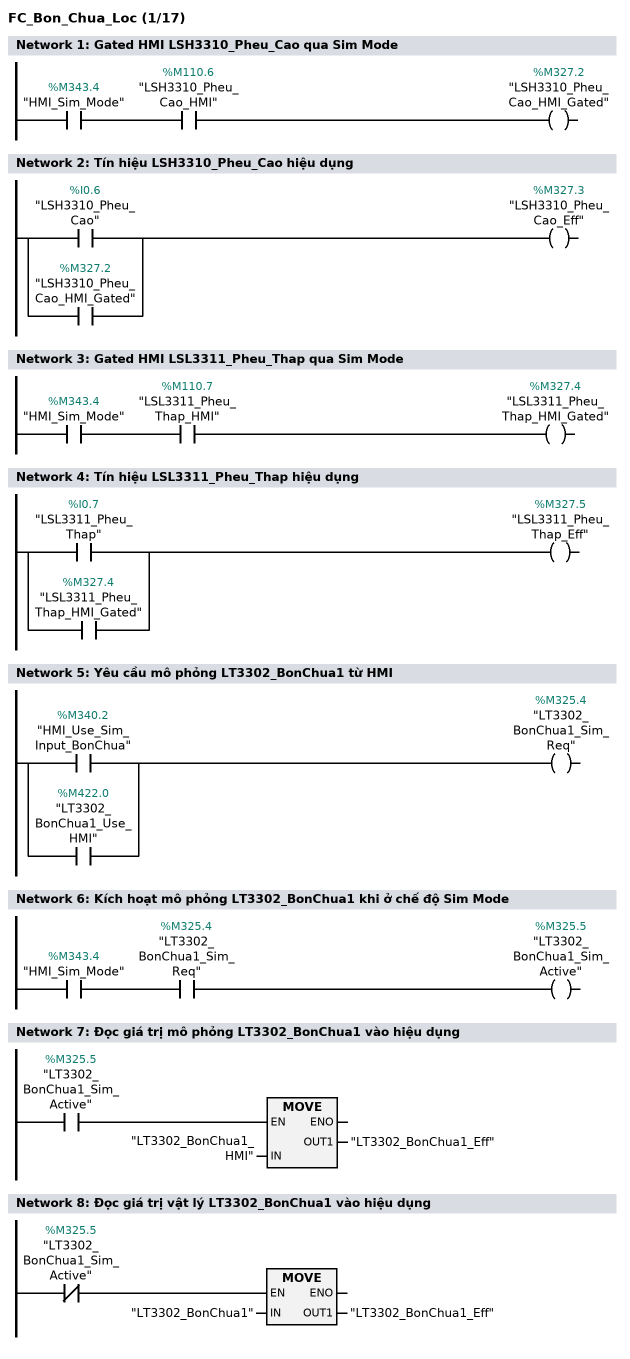
   RUNG wire#powerrail
      Contact( "HMI_Sim_Mode" )
      Contact( "LSH3310_Pheu_Cao_HMI" )
      Coil( "LSH3310_Pheu_Cao_HMI_Gated" )
   END_RUNG
   // the same network as SCL:
   "LSH3310_Pheu_Cao_HMI_Gated" := "HMI_Sim_Mode" AND "LSH3310_Pheu_Cao_HMI";
END_REGION

REGION Network 2: Tín hiệu LSH3310_Pheu_Cao hiệu dụng
   RUNG wire#powerrail
      Contact( "LSH3310_Pheu_Cao" )
      wire#w1
      Coil( "LSH3310_Pheu_Cao_Eff" )
   END_RUNG
   RUNG wire#powerrail
      Contact( "LSH3310_Pheu_Cao_HMI_Gated" )
   END_RUNG wire#w1
   // the same network as SCL:
   "LSH3310_Pheu_Cao_Eff" := "LSH3310_Pheu_Cao" OR "LSH3310_Pheu_Cao_HMI_Gated";
END_REGION

REGION Network 3: Gated HMI LSL3311_Pheu_Thap qua Sim Mode
   RUNG wire#powerrail
      Contact( "HMI_Sim_Mode" )
      Contact( "LSL3311_Pheu_Thap_HMI" )
      Coil( "LSL3311_Pheu_Thap_HMI_Gated" )
   END_RUNG
   // the same network as SCL:
   "LSL3311_Pheu_Thap_HMI_Gated" := "HMI_Sim_Mode" AND "LSL3311_Pheu_Thap_HMI";
END_REGION

REGION Network 4: Tín hiệu LSL3311_Pheu_Thap hiệu dụng
   RUNG wire#powerrail
      Contact( "LSL3311_Pheu_Thap" )
      wire#w1
      Coil( "LSL3311_Pheu_Thap_Eff" )
   END_RUNG
   RUNG wire#powerrail
      Contact( "LSL3311_Pheu_Thap_HMI_Gated" )
   END_RUNG wire#w1
   // the same network as SCL:
   "LSL3311_Pheu_Thap_Eff" := "LSL3311_Pheu_Thap" OR "LSL3311_Pheu_Thap_HMI_Gated";
END_REGION

REGION Network 5: Yêu cầu mô phỏng LT3302_BonChua1 từ HMI
   RUNG wire#powerrail
      Contact( "HMI_Use_Sim_Input_BonChua" )
      wire#w1
      Coil( "LT3302_BonChua1_Sim_Req" )
   END_RUNG
   RUNG wire#powerrail
      Contact( "LT3302_BonChua1_Use_HMI" )
   END_RUNG wire#w1
   // the same network as SCL:
   "LT3302_BonChua1_Sim_Req" := "HMI_Use_Sim_Input_BonChua" OR "LT3302_BonChua1_Use_HMI";
END_REGION

REGION Network 6: Kích hoạt mô phỏng LT3302_BonChua1 khi ở chế độ Sim Mode
   RUNG wire#powerrail
      Contact( "HMI_Sim_Mode" )
      Contact( "LT3302_BonChua1_Sim_Req" )
      Coil( "LT3302_BonChua1_Sim_Active" )
   END_RUNG
   // the same network as SCL:
   "LT3302_BonChua1_Sim_Active" := "HMI_Sim_Mode" AND "LT3302_BonChua1_Sim_Req";
END_REGION

REGION Network 7: Đọc giá trị mô phỏng LT3302_BonChua1 vào hiệu dụng
   RUNG wire#powerrail
      Contact( "LT3302_BonChua1_Sim_Active" )
      { S7_GenerateENO := "TRUE" } Move(in := "LT3302_BonChua1_HMI", out1 => "LT3302_BonChua1_Eff")
   END_RUNG
   // the same network as SCL:
   IF "LT3302_BonChua1_Sim_Active" THEN "LT3302_BonChua1_Eff" := "LT3302_BonChua1_HMI"; END_IF;
END_REGION

REGION Network 8: Đọc giá trị vật lý LT3302_BonChua1 vào hiệu dụng
   RUNG wire#powerrail
      I_Contact( "LT3302_BonChua1_Sim_Active" )
      { S7_GenerateENO := "TRUE" } Move(in := "LT3302_BonChua1", out1 => "LT3302_BonChua1_Eff")
   END_RUNG
   // the same network as SCL:
   IF NOT "LT3302_BonChua1_Sim_Active" THEN "LT3302_BonChua1_Eff" := "LT3302_BonChua1"; END_IF;
END_REGION

REGION Network 9: Yêu cầu mô phỏng TT3301_BonChua1 từ HMI
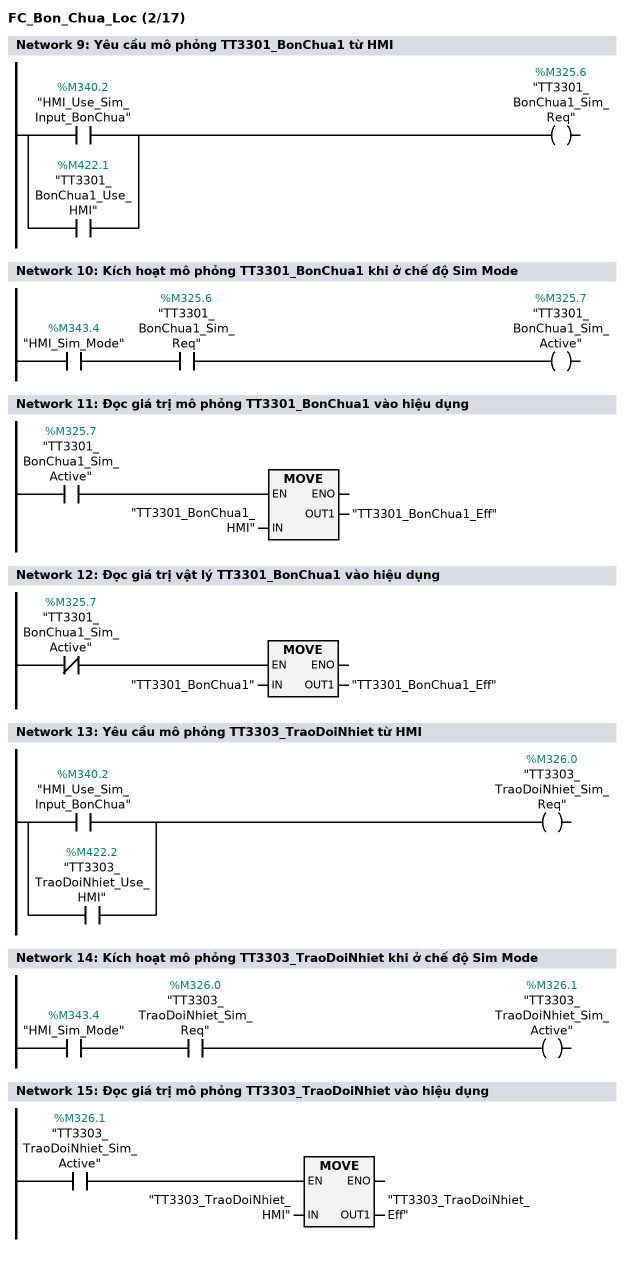
   RUNG wire#powerrail
      Contact( "HMI_Use_Sim_Input_BonChua" )
      wire#w1
      Coil( "TT3301_BonChua1_Sim_Req" )
   END_RUNG
   RUNG wire#powerrail
      Contact( "TT3301_BonChua1_Use_HMI" )
   END_RUNG wire#w1
   // the same network as SCL:
   "TT3301_BonChua1_Sim_Req" := "HMI_Use_Sim_Input_BonChua" OR "TT3301_BonChua1_Use_HMI";
END_REGION

REGION Network 10: Kích hoạt mô phỏng TT3301_BonChua1 khi ở chế độ Sim Mode
   RUNG wire#powerrail
      Contact( "HMI_Sim_Mode" )
      Contact( "TT3301_BonChua1_Sim_Req" )
      Coil( "TT3301_BonChua1_Sim_Active" )
   END_RUNG
   // the same network as SCL:
   "TT3301_BonChua1_Sim_Active" := "HMI_Sim_Mode" AND "TT3301_BonChua1_Sim_Req";
END_REGION

REGION Network 11: Đọc giá trị mô phỏng TT3301_BonChua1 vào hiệu dụng
   RUNG wire#powerrail
      Contact( "TT3301_BonChua1_Sim_Active" )
      { S7_GenerateENO := "TRUE" } Move(in := "TT3301_BonChua1_HMI", out1 => "TT3301_BonChua1_Eff")
   END_RUNG
   // the same network as SCL:
   IF "TT3301_BonChua1_Sim_Active" THEN "TT3301_BonChua1_Eff" := "TT3301_BonChua1_HMI"; END_IF;
END_REGION

REGION Network 12: Đọc giá trị vật lý TT3301_BonChua1 vào hiệu dụng
   RUNG wire#powerrail
      I_Contact( "TT3301_BonChua1_Sim_Active" )
      { S7_GenerateENO := "TRUE" } Move(in := "TT3301_BonChua1", out1 => "TT3301_BonChua1_Eff")
   END_RUNG
   // the same network as SCL:
   IF NOT "TT3301_BonChua1_Sim_Active" THEN "TT3301_BonChua1_Eff" := "TT3301_BonChua1"; END_IF;
END_REGION

REGION Network 13: Yêu cầu mô phỏng TT3303_TraoDoiNhiet từ HMI
   RUNG wire#powerrail
      Contact( "HMI_Use_Sim_Input_BonChua" )
      wire#w1
      Coil( "TT3303_TraoDoiNhiet_Sim_Req" )
   END_RUNG
   RUNG wire#powerrail
      Contact( "TT3303_TraoDoiNhiet_Use_HMI" )
   END_RUNG wire#w1
   // the same network as SCL:
   "TT3303_TraoDoiNhiet_Sim_Req" := "HMI_Use_Sim_Input_BonChua" OR "TT3303_TraoDoiNhiet_Use_HMI";
END_REGION

REGION Network 14: Kích hoạt mô phỏng TT3303_TraoDoiNhiet khi ở chế độ Sim Mode
   RUNG wire#powerrail
      Contact( "HMI_Sim_Mode" )
      Contact( "TT3303_TraoDoiNhiet_Sim_Req" )
      Coil( "TT3303_TraoDoiNhiet_Sim_Active" )
   END_RUNG
   // the same network as SCL:
   "TT3303_TraoDoiNhiet_Sim_Active" := "HMI_Sim_Mode" AND "TT3303_TraoDoiNhiet_Sim_Req";
END_REGION

REGION Network 15: Đọc giá trị mô phỏng TT3303_TraoDoiNhiet vào hiệu dụng
   RUNG wire#powerrail
      Contact( "TT3303_TraoDoiNhiet_Sim_Active" )
      { S7_GenerateENO := "TRUE" } Move(in := "TT3303_TraoDoiNhiet_HMI", out1 => "TT3303_TraoDoiNhiet_Eff")
   END_RUNG
   // the same network as SCL:
   IF "TT3303_TraoDoiNhiet_Sim_Active" THEN "TT3303_TraoDoiNhiet_Eff" := "TT3303_TraoDoiNhiet_HMI"; END_IF;
END_REGION

REGION Network 16: Đọc giá trị vật lý TT3303_TraoDoiNhiet vào hiệu dụng
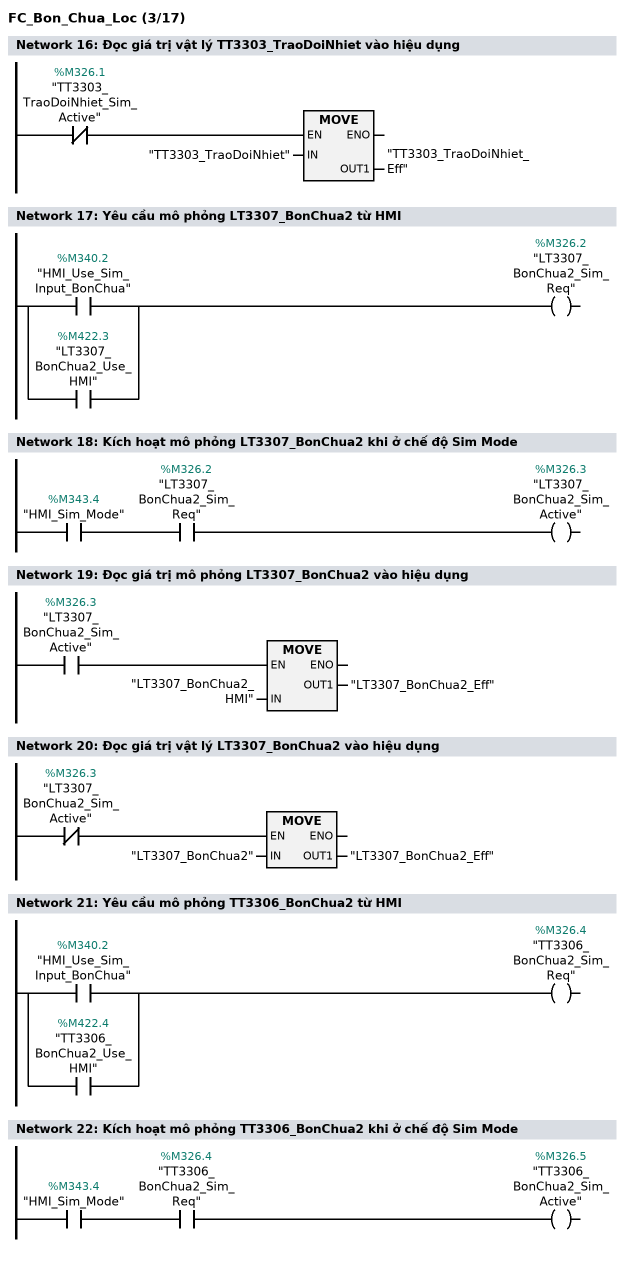
   RUNG wire#powerrail
      I_Contact( "TT3303_TraoDoiNhiet_Sim_Active" )
      { S7_GenerateENO := "TRUE" } Move(in := "TT3303_TraoDoiNhiet", out1 => "TT3303_TraoDoiNhiet_Eff")
   END_RUNG
   // the same network as SCL:
   IF NOT "TT3303_TraoDoiNhiet_Sim_Active" THEN "TT3303_TraoDoiNhiet_Eff" := "TT3303_TraoDoiNhiet"; END_IF;
END_REGION

REGION Network 17: Yêu cầu mô phỏng LT3307_BonChua2 từ HMI
   RUNG wire#powerrail
      Contact( "HMI_Use_Sim_Input_BonChua" )
      wire#w1
      Coil( "LT3307_BonChua2_Sim_Req" )
   END_RUNG
   RUNG wire#powerrail
      Contact( "LT3307_BonChua2_Use_HMI" )
   END_RUNG wire#w1
   // the same network as SCL:
   "LT3307_BonChua2_Sim_Req" := "HMI_Use_Sim_Input_BonChua" OR "LT3307_BonChua2_Use_HMI";
END_REGION

REGION Network 18: Kích hoạt mô phỏng LT3307_BonChua2 khi ở chế độ Sim Mode
   RUNG wire#powerrail
      Contact( "HMI_Sim_Mode" )
      Contact( "LT3307_BonChua2_Sim_Req" )
      Coil( "LT3307_BonChua2_Sim_Active" )
   END_RUNG
   // the same network as SCL:
   "LT3307_BonChua2_Sim_Active" := "HMI_Sim_Mode" AND "LT3307_BonChua2_Sim_Req";
END_REGION

REGION Network 19: Đọc giá trị mô phỏng LT3307_BonChua2 vào hiệu dụng
   RUNG wire#powerrail
      Contact( "LT3307_BonChua2_Sim_Active" )
      { S7_GenerateENO := "TRUE" } Move(in := "LT3307_BonChua2_HMI", out1 => "LT3307_BonChua2_Eff")
   END_RUNG
   // the same network as SCL:
   IF "LT3307_BonChua2_Sim_Active" THEN "LT3307_BonChua2_Eff" := "LT3307_BonChua2_HMI"; END_IF;
END_REGION

REGION Network 20: Đọc giá trị vật lý LT3307_BonChua2 vào hiệu dụng
   RUNG wire#powerrail
      I_Contact( "LT3307_BonChua2_Sim_Active" )
      { S7_GenerateENO := "TRUE" } Move(in := "LT3307_BonChua2", out1 => "LT3307_BonChua2_Eff")
   END_RUNG
   // the same network as SCL:
   IF NOT "LT3307_BonChua2_Sim_Active" THEN "LT3307_BonChua2_Eff" := "LT3307_BonChua2"; END_IF;
END_REGION

REGION Network 21: Yêu cầu mô phỏng TT3306_BonChua2 từ HMI
   RUNG wire#powerrail
      Contact( "HMI_Use_Sim_Input_BonChua" )
      wire#w1
      Coil( "TT3306_BonChua2_Sim_Req" )
   END_RUNG
   RUNG wire#powerrail
      Contact( "TT3306_BonChua2_Use_HMI" )
   END_RUNG wire#w1
   // the same network as SCL:
   "TT3306_BonChua2_Sim_Req" := "HMI_Use_Sim_Input_BonChua" OR "TT3306_BonChua2_Use_HMI";
END_REGION

REGION Network 22: Kích hoạt mô phỏng TT3306_BonChua2 khi ở chế độ Sim Mode
   RUNG wire#powerrail
      Contact( "HMI_Sim_Mode" )
      Contact( "TT3306_BonChua2_Sim_Req" )
      Coil( "TT3306_BonChua2_Sim_Active" )
   END_RUNG
   // the same network as SCL:
   "TT3306_BonChua2_Sim_Active" := "HMI_Sim_Mode" AND "TT3306_BonChua2_Sim_Req";
END_REGION

REGION Network 23: Đọc giá trị mô phỏng TT3306_BonChua2 vào hiệu dụng
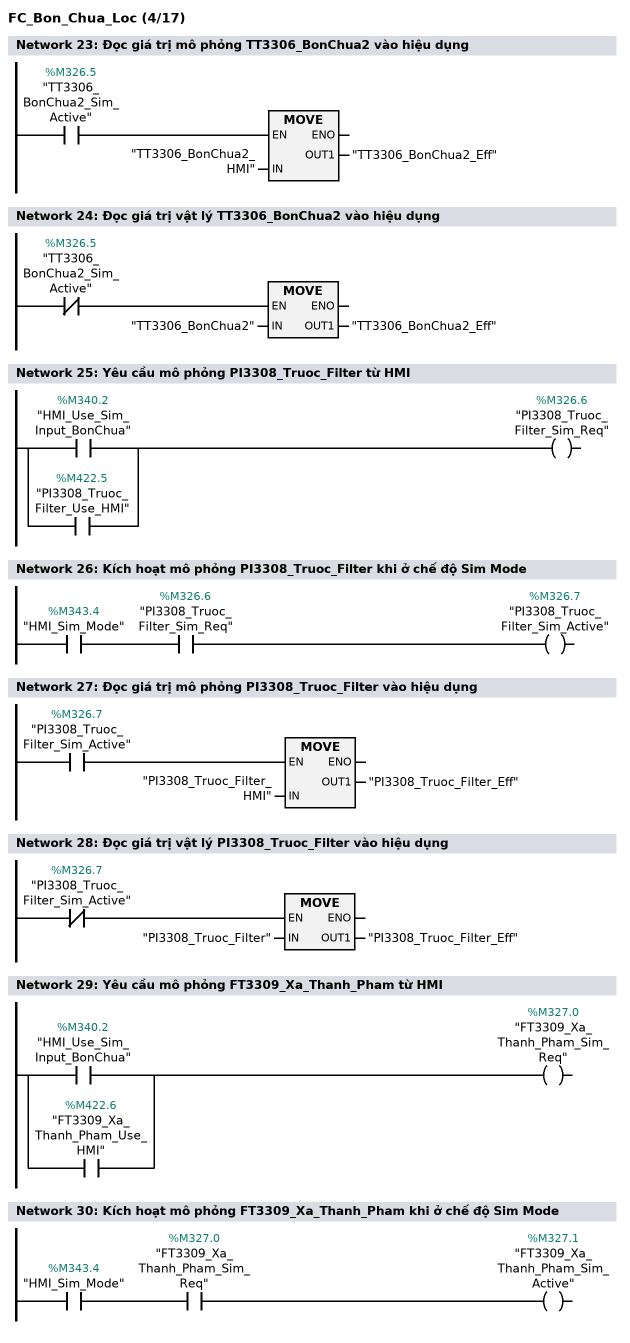
   RUNG wire#powerrail
      Contact( "TT3306_BonChua2_Sim_Active" )
      { S7_GenerateENO := "TRUE" } Move(in := "TT3306_BonChua2_HMI", out1 => "TT3306_BonChua2_Eff")
   END_RUNG
   // the same network as SCL:
   IF "TT3306_BonChua2_Sim_Active" THEN "TT3306_BonChua2_Eff" := "TT3306_BonChua2_HMI"; END_IF;
END_REGION

REGION Network 24: Đọc giá trị vật lý TT3306_BonChua2 vào hiệu dụng
   RUNG wire#powerrail
      I_Contact( "TT3306_BonChua2_Sim_Active" )
      { S7_GenerateENO := "TRUE" } Move(in := "TT3306_BonChua2", out1 => "TT3306_BonChua2_Eff")
   END_RUNG
   // the same network as SCL:
   IF NOT "TT3306_BonChua2_Sim_Active" THEN "TT3306_BonChua2_Eff" := "TT3306_BonChua2"; END_IF;
END_REGION

REGION Network 25: Yêu cầu mô phỏng PI3308_Truoc_Filter từ HMI
   RUNG wire#powerrail
      Contact( "HMI_Use_Sim_Input_BonChua" )
      wire#w1
      Coil( "PI3308_Truoc_Filter_Sim_Req" )
   END_RUNG
   RUNG wire#powerrail
      Contact( "PI3308_Truoc_Filter_Use_HMI" )
   END_RUNG wire#w1
   // the same network as SCL:
   "PI3308_Truoc_Filter_Sim_Req" := "HMI_Use_Sim_Input_BonChua" OR "PI3308_Truoc_Filter_Use_HMI";
END_REGION

REGION Network 26: Kích hoạt mô phỏng PI3308_Truoc_Filter khi ở chế độ Sim Mode
   RUNG wire#powerrail
      Contact( "HMI_Sim_Mode" )
      Contact( "PI3308_Truoc_Filter_Sim_Req" )
      Coil( "PI3308_Truoc_Filter_Sim_Active" )
   END_RUNG
   // the same network as SCL:
   "PI3308_Truoc_Filter_Sim_Active" := "HMI_Sim_Mode" AND "PI3308_Truoc_Filter_Sim_Req";
END_REGION

REGION Network 27: Đọc giá trị mô phỏng PI3308_Truoc_Filter vào hiệu dụng
   RUNG wire#powerrail
      Contact( "PI3308_Truoc_Filter_Sim_Active" )
      { S7_GenerateENO := "TRUE" } Move(in := "PI3308_Truoc_Filter_HMI", out1 => "PI3308_Truoc_Filter_Eff")
   END_RUNG
   // the same network as SCL:
   IF "PI3308_Truoc_Filter_Sim_Active" THEN "PI3308_Truoc_Filter_Eff" := "PI3308_Truoc_Filter_HMI"; END_IF;
END_REGION

REGION Network 28: Đọc giá trị vật lý PI3308_Truoc_Filter vào hiệu dụng
   RUNG wire#powerrail
      I_Contact( "PI3308_Truoc_Filter_Sim_Active" )
      { S7_GenerateENO := "TRUE" } Move(in := "PI3308_Truoc_Filter", out1 => "PI3308_Truoc_Filter_Eff")
   END_RUNG
   // the same network as SCL:
   IF NOT "PI3308_Truoc_Filter_Sim_Active" THEN "PI3308_Truoc_Filter_Eff" := "PI3308_Truoc_Filter"; END_IF;
END_REGION

REGION Network 29: Yêu cầu mô phỏng FT3309_Xa_Thanh_Pham từ HMI
   RUNG wire#powerrail
      Contact( "HMI_Use_Sim_Input_BonChua" )
      wire#w1
      Coil( "FT3309_Xa_Thanh_Pham_Sim_Req" )
   END_RUNG
   RUNG wire#powerrail
      Contact( "FT3309_Xa_Thanh_Pham_Use_HMI" )
   END_RUNG wire#w1
   // the same network as SCL:
   "FT3309_Xa_Thanh_Pham_Sim_Req" := "HMI_Use_Sim_Input_BonChua" OR "FT3309_Xa_Thanh_Pham_Use_HMI";
END_REGION

REGION Network 30: Kích hoạt mô phỏng FT3309_Xa_Thanh_Pham khi ở chế độ Sim Mode
   RUNG wire#powerrail
      Contact( "HMI_Sim_Mode" )
      Contact( "FT3309_Xa_Thanh_Pham_Sim_Req" )
      Coil( "FT3309_Xa_Thanh_Pham_Sim_Active" )
   END_RUNG
   // the same network as SCL:
   "FT3309_Xa_Thanh_Pham_Sim_Active" := "HMI_Sim_Mode" AND "FT3309_Xa_Thanh_Pham_Sim_Req";
END_REGION

REGION Network 31: Đọc giá trị mô phỏng FT3309_Xa_Thanh_Pham vào hiệu dụng
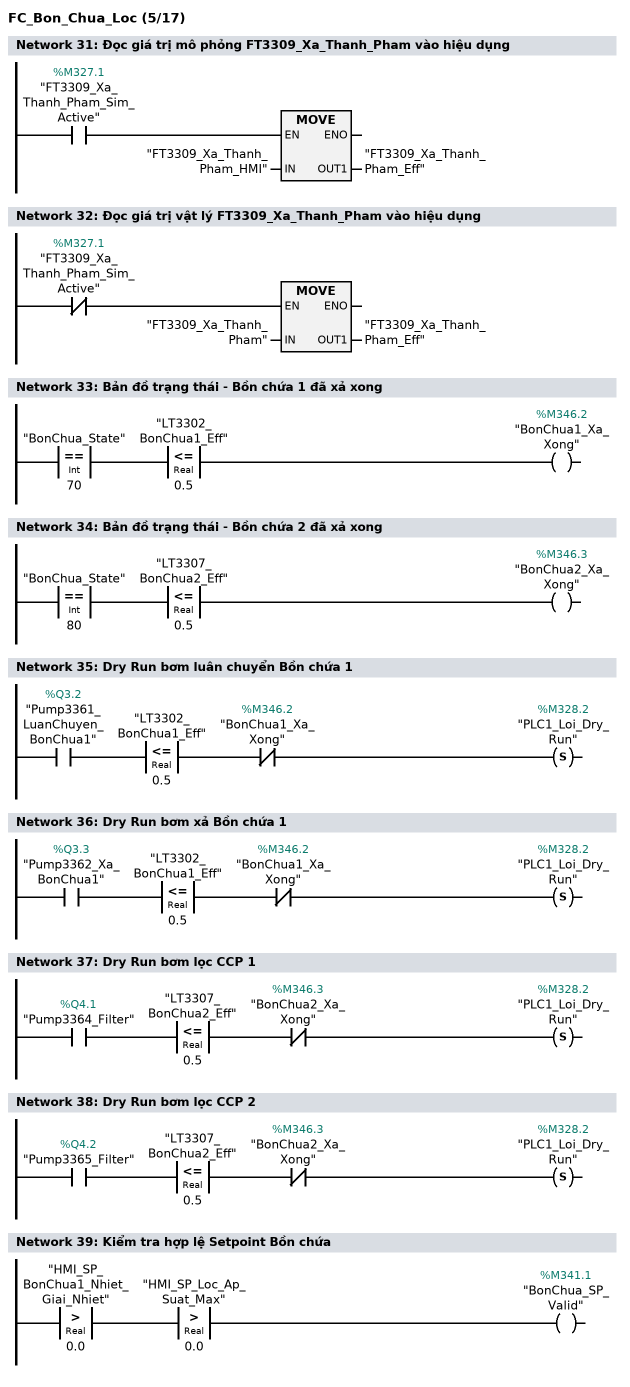
   RUNG wire#powerrail
      Contact( "FT3309_Xa_Thanh_Pham_Sim_Active" )
      { S7_GenerateENO := "TRUE" } Move(in := "FT3309_Xa_Thanh_Pham_HMI", out1 => "FT3309_Xa_Thanh_Pham_Eff")
   END_RUNG
   // the same network as SCL:
   IF "FT3309_Xa_Thanh_Pham_Sim_Active" THEN
       "FT3309_Xa_Thanh_Pham_Eff" := "FT3309_Xa_Thanh_Pham_HMI";
   END_IF;
END_REGION

REGION Network 32: Đọc giá trị vật lý FT3309_Xa_Thanh_Pham vào hiệu dụng
   RUNG wire#powerrail
      I_Contact( "FT3309_Xa_Thanh_Pham_Sim_Active" )
      { S7_GenerateENO := "TRUE" } Move(in := "FT3309_Xa_Thanh_Pham", out1 => "FT3309_Xa_Thanh_Pham_Eff")
   END_RUNG
   // the same network as SCL:
   IF NOT "FT3309_Xa_Thanh_Pham_Sim_Active" THEN
       "FT3309_Xa_Thanh_Pham_Eff" := "FT3309_Xa_Thanh_Pham";
   END_IF;
END_REGION

REGION Network 33: Bản đồ trạng thái - Bồn chứa 1 đã xả xong
   RUNG wire#powerrail
      { S7_Templates := "SrcType := Int" } EQ_Contact(in1 := "BonChua_State", in2 := 70)
      { S7_Templates := "SrcType := Real" } LE_Contact(in1 := "LT3302_BonChua1_Eff", in2 := 0.5)
      Coil( "BonChua1_Xa_Xong" )
   END_RUNG
   // the same network as SCL:
   "BonChua1_Xa_Xong" := ("BonChua_State" = 70) AND ("LT3302_BonChua1_Eff" <= 0.5);
END_REGION

REGION Network 34: Bản đồ trạng thái - Bồn chứa 2 đã xả xong
   RUNG wire#powerrail
      { S7_Templates := "SrcType := Int" } EQ_Contact(in1 := "BonChua_State", in2 := 80)
      { S7_Templates := "SrcType := Real" } LE_Contact(in1 := "LT3307_BonChua2_Eff", in2 := 0.5)
      Coil( "BonChua2_Xa_Xong" )
   END_RUNG
   // the same network as SCL:
   "BonChua2_Xa_Xong" := ("BonChua_State" = 80) AND ("LT3307_BonChua2_Eff" <= 0.5);
END_REGION

REGION Network 35: Dry Run bơm luân chuyển Bồn chứa 1
   RUNG wire#powerrail
      Contact( "Pump3361_LuanChuyen_BonChua1" )
      { S7_Templates := "SrcType := Real" } LE_Contact(in1 := "LT3302_BonChua1_Eff", in2 := 0.5)
      I_Contact( "BonChua1_Xa_Xong" )
      S_Coil( "PLC1_Loi_Dry_Run" )
   END_RUNG
   // the same network as SCL:
   IF "Pump3361_LuanChuyen_BonChua1" AND ("LT3302_BonChua1_Eff" <= 0.5) AND NOT "BonChua1_Xa_Xong" THEN
       "PLC1_Loi_Dry_Run" := TRUE;
   END_IF;
END_REGION

REGION Network 36: Dry Run bơm xả Bồn chứa 1
   RUNG wire#powerrail
      Contact( "Pump3362_Xa_BonChua1" )
      { S7_Templates := "SrcType := Real" } LE_Contact(in1 := "LT3302_BonChua1_Eff", in2 := 0.5)
      I_Contact( "BonChua1_Xa_Xong" )
      S_Coil( "PLC1_Loi_Dry_Run" )
   END_RUNG
   // the same network as SCL:
   IF "Pump3362_Xa_BonChua1" AND ("LT3302_BonChua1_Eff" <= 0.5) AND NOT "BonChua1_Xa_Xong" THEN
       "PLC1_Loi_Dry_Run" := TRUE;
   END_IF;
END_REGION

REGION Network 37: Dry Run bơm lọc CCP 1
   RUNG wire#powerrail
      Contact( "Pump3364_Filter" )
      { S7_Templates := "SrcType := Real" } LE_Contact(in1 := "LT3307_BonChua2_Eff", in2 := 0.5)
      I_Contact( "BonChua2_Xa_Xong" )
      S_Coil( "PLC1_Loi_Dry_Run" )
   END_RUNG
   // the same network as SCL:
   IF "Pump3364_Filter" AND ("LT3307_BonChua2_Eff" <= 0.5) AND NOT "BonChua2_Xa_Xong" THEN
       "PLC1_Loi_Dry_Run" := TRUE;
   END_IF;
END_REGION

REGION Network 38: Dry Run bơm lọc CCP 2
   RUNG wire#powerrail
      Contact( "Pump3365_Filter" )
      { S7_Templates := "SrcType := Real" } LE_Contact(in1 := "LT3307_BonChua2_Eff", in2 := 0.5)
      I_Contact( "BonChua2_Xa_Xong" )
      S_Coil( "PLC1_Loi_Dry_Run" )
   END_RUNG
   // the same network as SCL:
   IF "Pump3365_Filter" AND ("LT3307_BonChua2_Eff" <= 0.5) AND NOT "BonChua2_Xa_Xong" THEN
       "PLC1_Loi_Dry_Run" := TRUE;
   END_IF;
END_REGION

REGION Network 39: Kiểm tra hợp lệ Setpoint Bồn chứa
   RUNG wire#powerrail
      { S7_Templates := "SrcType := Real" } GT_Contact(in1 := "HMI_SP_BonChua1_Nhiet_Giai_Nhiet", in2 := 0.0)
      { S7_Templates := "SrcType := Real" } GT_Contact(in1 := "HMI_SP_Loc_Ap_Suat_Max", in2 := 0.0)
      Coil( "BonChua_SP_Valid" )
   END_RUNG
   // the same network as SCL:
   "BonChua_SP_Valid" := ("HMI_SP_BonChua1_Nhiet_Giai_Nhiet" > 0.0) AND ("HMI_SP_Loc_Ap_Suat_Max" > 0.0);
END_REGION

REGION Network 40: Stop hoặc Lỗi tổng - reset BonChua_Step_Nhan_Dich
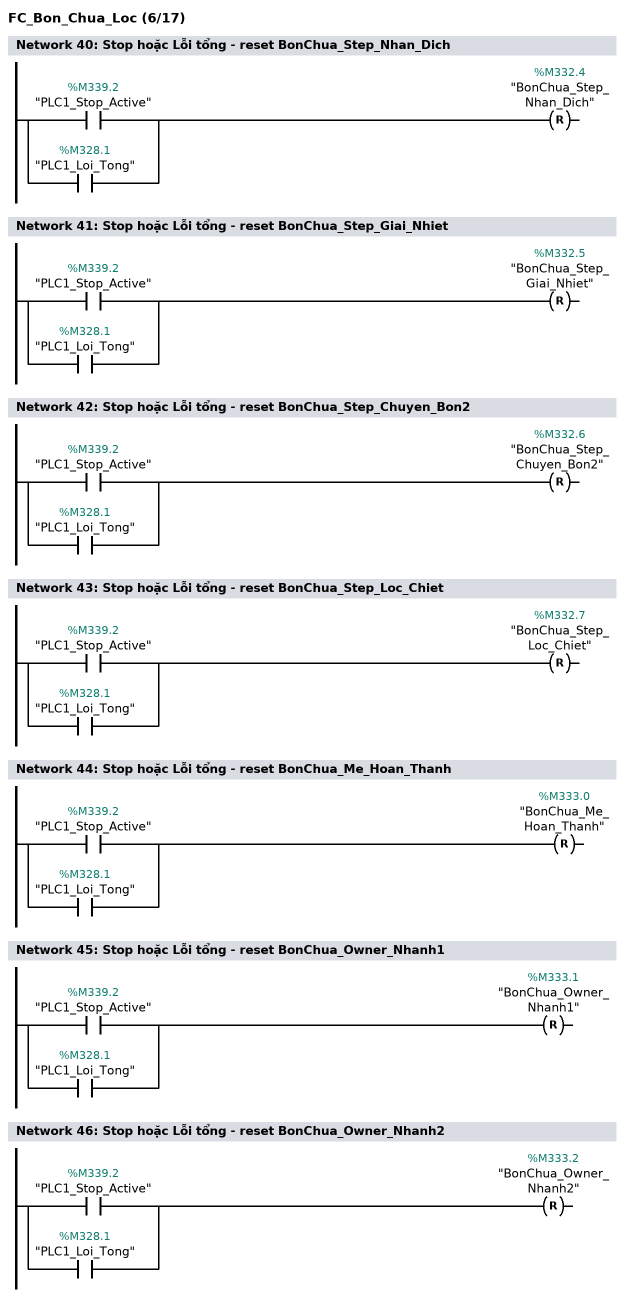
   RUNG wire#powerrail
      Contact( "PLC1_Stop_Active" )
      wire#w1
      R_Coil( "BonChua_Step_Nhan_Dich" )
   END_RUNG
   RUNG wire#powerrail
      Contact( "PLC1_Loi_Tong" )
   END_RUNG wire#w1
   // the same network as SCL:
   IF "PLC1_Stop_Active" OR "PLC1_Loi_Tong" THEN "BonChua_Step_Nhan_Dich" := FALSE; END_IF;
END_REGION

REGION Network 41: Stop hoặc Lỗi tổng - reset BonChua_Step_Giai_Nhiet
   RUNG wire#powerrail
      Contact( "PLC1_Stop_Active" )
      wire#w1
      R_Coil( "BonChua_Step_Giai_Nhiet" )
   END_RUNG
   RUNG wire#powerrail
      Contact( "PLC1_Loi_Tong" )
   END_RUNG wire#w1
   // the same network as SCL:
   IF "PLC1_Stop_Active" OR "PLC1_Loi_Tong" THEN "BonChua_Step_Giai_Nhiet" := FALSE; END_IF;
END_REGION

REGION Network 42: Stop hoặc Lỗi tổng - reset BonChua_Step_Chuyen_Bon2
   RUNG wire#powerrail
      Contact( "PLC1_Stop_Active" )
      wire#w1
      R_Coil( "BonChua_Step_Chuyen_Bon2" )
   END_RUNG
   RUNG wire#powerrail
      Contact( "PLC1_Loi_Tong" )
   END_RUNG wire#w1
   // the same network as SCL:
   IF "PLC1_Stop_Active" OR "PLC1_Loi_Tong" THEN "BonChua_Step_Chuyen_Bon2" := FALSE; END_IF;
END_REGION

REGION Network 43: Stop hoặc Lỗi tổng - reset BonChua_Step_Loc_Chiet
   RUNG wire#powerrail
      Contact( "PLC1_Stop_Active" )
      wire#w1
      R_Coil( "BonChua_Step_Loc_Chiet" )
   END_RUNG
   RUNG wire#powerrail
      Contact( "PLC1_Loi_Tong" )
   END_RUNG wire#w1
   // the same network as SCL:
   IF "PLC1_Stop_Active" OR "PLC1_Loi_Tong" THEN "BonChua_Step_Loc_Chiet" := FALSE; END_IF;
END_REGION

REGION Network 44: Stop hoặc Lỗi tổng - reset BonChua_Me_Hoan_Thanh
   RUNG wire#powerrail
      Contact( "PLC1_Stop_Active" )
      wire#w1
      R_Coil( "BonChua_Me_Hoan_Thanh" )
   END_RUNG
   RUNG wire#powerrail
      Contact( "PLC1_Loi_Tong" )
   END_RUNG wire#w1
   // the same network as SCL:
   IF "PLC1_Stop_Active" OR "PLC1_Loi_Tong" THEN "BonChua_Me_Hoan_Thanh" := FALSE; END_IF;
END_REGION

REGION Network 45: Stop hoặc Lỗi tổng - reset BonChua_Owner_Nhanh1
   RUNG wire#powerrail
      Contact( "PLC1_Stop_Active" )
      wire#w1
      R_Coil( "BonChua_Owner_Nhanh1" )
   END_RUNG
   RUNG wire#powerrail
      Contact( "PLC1_Loi_Tong" )
   END_RUNG wire#w1
   // the same network as SCL:
   IF "PLC1_Stop_Active" OR "PLC1_Loi_Tong" THEN "BonChua_Owner_Nhanh1" := FALSE; END_IF;
END_REGION

REGION Network 46: Stop hoặc Lỗi tổng - reset BonChua_Owner_Nhanh2
   RUNG wire#powerrail
      Contact( "PLC1_Stop_Active" )
      wire#w1
      R_Coil( "BonChua_Owner_Nhanh2" )
   END_RUNG
   RUNG wire#powerrail
      Contact( "PLC1_Loi_Tong" )
   END_RUNG wire#w1
   // the same network as SCL:
   IF "PLC1_Stop_Active" OR "PLC1_Loi_Tong" THEN "BonChua_Owner_Nhanh2" := FALSE; END_IF;
END_REGION

REGION Network 47: Stop hoặc Lỗi tổng - reset V3331_Xa_BonChua1
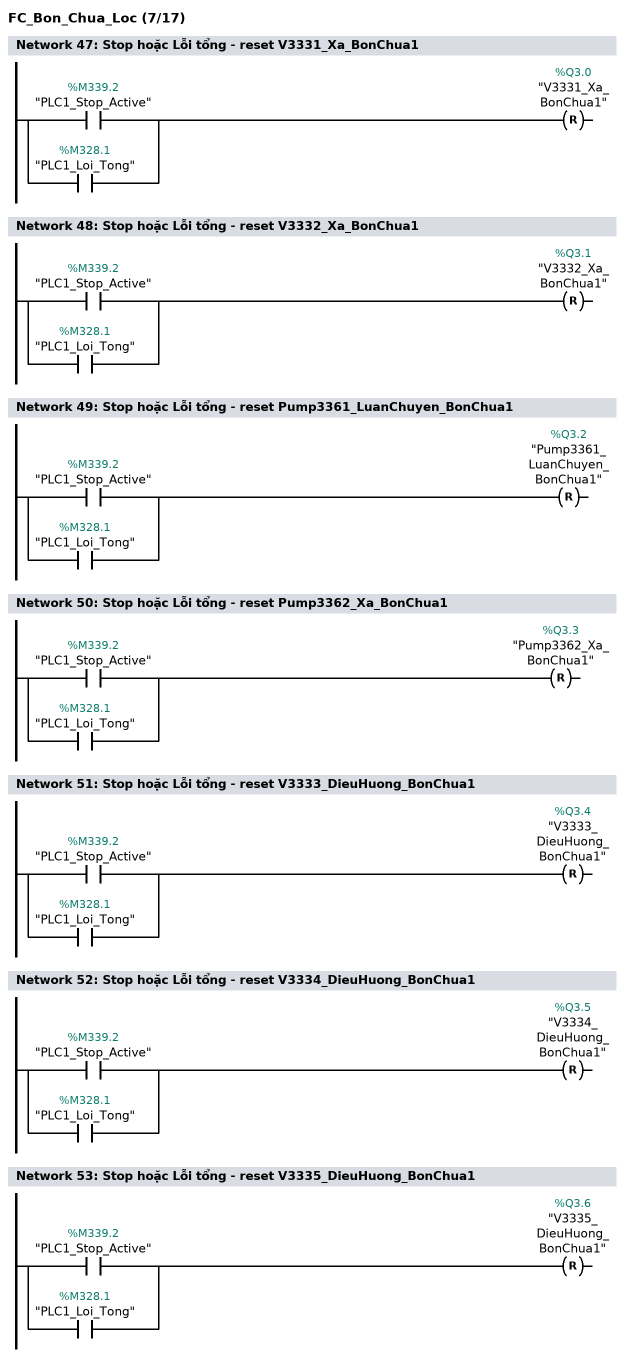
   RUNG wire#powerrail
      Contact( "PLC1_Stop_Active" )
      wire#w1
      R_Coil( "V3331_Xa_BonChua1" )
   END_RUNG
   RUNG wire#powerrail
      Contact( "PLC1_Loi_Tong" )
   END_RUNG wire#w1
   // the same network as SCL:
   IF "PLC1_Stop_Active" OR "PLC1_Loi_Tong" THEN "V3331_Xa_BonChua1" := FALSE; END_IF;
END_REGION

REGION Network 48: Stop hoặc Lỗi tổng - reset V3332_Xa_BonChua1
   RUNG wire#powerrail
      Contact( "PLC1_Stop_Active" )
      wire#w1
      R_Coil( "V3332_Xa_BonChua1" )
   END_RUNG
   RUNG wire#powerrail
      Contact( "PLC1_Loi_Tong" )
   END_RUNG wire#w1
   // the same network as SCL:
   IF "PLC1_Stop_Active" OR "PLC1_Loi_Tong" THEN "V3332_Xa_BonChua1" := FALSE; END_IF;
END_REGION

REGION Network 49: Stop hoặc Lỗi tổng - reset Pump3361_LuanChuyen_BonChua1
   RUNG wire#powerrail
      Contact( "PLC1_Stop_Active" )
      wire#w1
      R_Coil( "Pump3361_LuanChuyen_BonChua1" )
   END_RUNG
   RUNG wire#powerrail
      Contact( "PLC1_Loi_Tong" )
   END_RUNG wire#w1
   // the same network as SCL:
   IF "PLC1_Stop_Active" OR "PLC1_Loi_Tong" THEN "Pump3361_LuanChuyen_BonChua1" := FALSE; END_IF;
END_REGION

REGION Network 50: Stop hoặc Lỗi tổng - reset Pump3362_Xa_BonChua1
   RUNG wire#powerrail
      Contact( "PLC1_Stop_Active" )
      wire#w1
      R_Coil( "Pump3362_Xa_BonChua1" )
   END_RUNG
   RUNG wire#powerrail
      Contact( "PLC1_Loi_Tong" )
   END_RUNG wire#w1
   // the same network as SCL:
   IF "PLC1_Stop_Active" OR "PLC1_Loi_Tong" THEN "Pump3362_Xa_BonChua1" := FALSE; END_IF;
END_REGION

REGION Network 51: Stop hoặc Lỗi tổng - reset V3333_DieuHuong_BonChua1
   RUNG wire#powerrail
      Contact( "PLC1_Stop_Active" )
      wire#w1
      R_Coil( "V3333_DieuHuong_BonChua1" )
   END_RUNG
   RUNG wire#powerrail
      Contact( "PLC1_Loi_Tong" )
   END_RUNG wire#w1
   // the same network as SCL:
   IF "PLC1_Stop_Active" OR "PLC1_Loi_Tong" THEN "V3333_DieuHuong_BonChua1" := FALSE; END_IF;
END_REGION

REGION Network 52: Stop hoặc Lỗi tổng - reset V3334_DieuHuong_BonChua1
   RUNG wire#powerrail
      Contact( "PLC1_Stop_Active" )
      wire#w1
      R_Coil( "V3334_DieuHuong_BonChua1" )
   END_RUNG
   RUNG wire#powerrail
      Contact( "PLC1_Loi_Tong" )
   END_RUNG wire#w1
   // the same network as SCL:
   IF "PLC1_Stop_Active" OR "PLC1_Loi_Tong" THEN "V3334_DieuHuong_BonChua1" := FALSE; END_IF;
END_REGION

REGION Network 53: Stop hoặc Lỗi tổng - reset V3335_DieuHuong_BonChua1
   RUNG wire#powerrail
      Contact( "PLC1_Stop_Active" )
      wire#w1
      R_Coil( "V3335_DieuHuong_BonChua1" )
   END_RUNG
   RUNG wire#powerrail
      Contact( "PLC1_Loi_Tong" )
   END_RUNG wire#w1
   // the same network as SCL:
   IF "PLC1_Stop_Active" OR "PLC1_Loi_Tong" THEN "V3335_DieuHuong_BonChua1" := FALSE; END_IF;
END_REGION

REGION Network 54: Stop hoặc Lỗi tổng - reset V3338_Xa_BonChua2
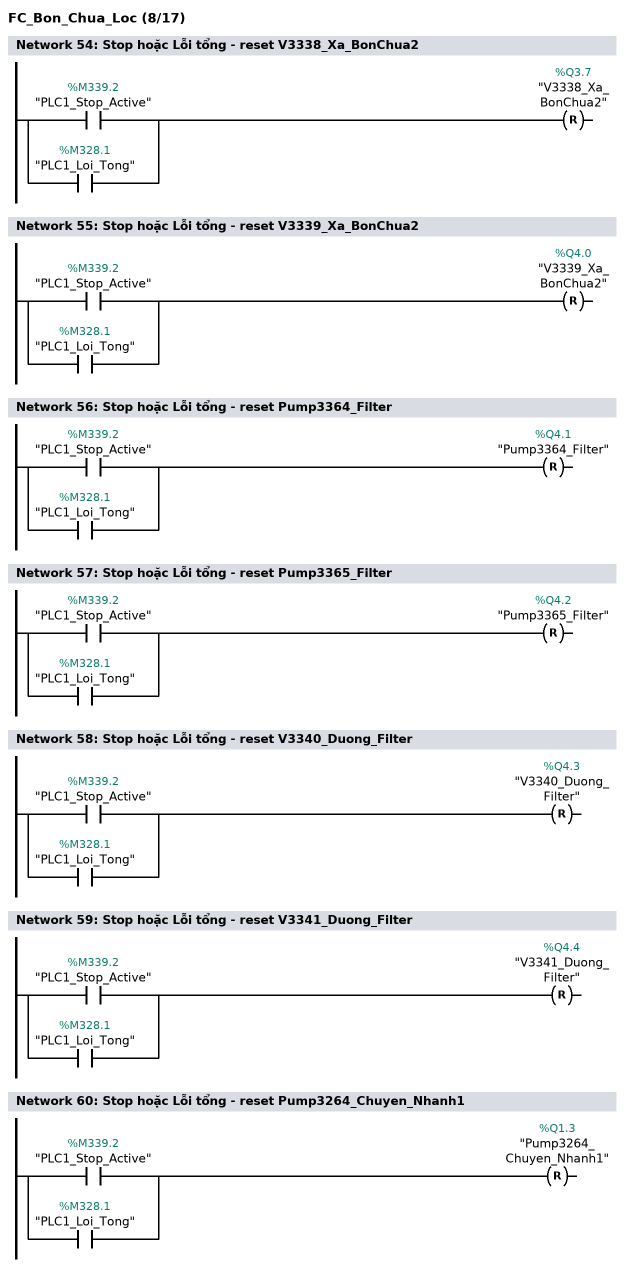
   RUNG wire#powerrail
      Contact( "PLC1_Stop_Active" )
      wire#w1
      R_Coil( "V3338_Xa_BonChua2" )
   END_RUNG
   RUNG wire#powerrail
      Contact( "PLC1_Loi_Tong" )
   END_RUNG wire#w1
   // the same network as SCL:
   IF "PLC1_Stop_Active" OR "PLC1_Loi_Tong" THEN "V3338_Xa_BonChua2" := FALSE; END_IF;
END_REGION

REGION Network 55: Stop hoặc Lỗi tổng - reset V3339_Xa_BonChua2
   RUNG wire#powerrail
      Contact( "PLC1_Stop_Active" )
      wire#w1
      R_Coil( "V3339_Xa_BonChua2" )
   END_RUNG
   RUNG wire#powerrail
      Contact( "PLC1_Loi_Tong" )
   END_RUNG wire#w1
   // the same network as SCL:
   IF "PLC1_Stop_Active" OR "PLC1_Loi_Tong" THEN "V3339_Xa_BonChua2" := FALSE; END_IF;
END_REGION

REGION Network 56: Stop hoặc Lỗi tổng - reset Pump3364_Filter
   RUNG wire#powerrail
      Contact( "PLC1_Stop_Active" )
      wire#w1
      R_Coil( "Pump3364_Filter" )
   END_RUNG
   RUNG wire#powerrail
      Contact( "PLC1_Loi_Tong" )
   END_RUNG wire#w1
   // the same network as SCL:
   IF "PLC1_Stop_Active" OR "PLC1_Loi_Tong" THEN "Pump3364_Filter" := FALSE; END_IF;
END_REGION

REGION Network 57: Stop hoặc Lỗi tổng - reset Pump3365_Filter
   RUNG wire#powerrail
      Contact( "PLC1_Stop_Active" )
      wire#w1
      R_Coil( "Pump3365_Filter" )
   END_RUNG
   RUNG wire#powerrail
      Contact( "PLC1_Loi_Tong" )
   END_RUNG wire#w1
   // the same network as SCL:
   IF "PLC1_Stop_Active" OR "PLC1_Loi_Tong" THEN "Pump3365_Filter" := FALSE; END_IF;
END_REGION

REGION Network 58: Stop hoặc Lỗi tổng - reset V3340_Duong_Filter
   RUNG wire#powerrail
      Contact( "PLC1_Stop_Active" )
      wire#w1
      R_Coil( "V3340_Duong_Filter" )
   END_RUNG
   RUNG wire#powerrail
      Contact( "PLC1_Loi_Tong" )
   END_RUNG wire#w1
   // the same network as SCL:
   IF "PLC1_Stop_Active" OR "PLC1_Loi_Tong" THEN "V3340_Duong_Filter" := FALSE; END_IF;
END_REGION

REGION Network 59: Stop hoặc Lỗi tổng - reset V3341_Duong_Filter
   RUNG wire#powerrail
      Contact( "PLC1_Stop_Active" )
      wire#w1
      R_Coil( "V3341_Duong_Filter" )
   END_RUNG
   RUNG wire#powerrail
      Contact( "PLC1_Loi_Tong" )
   END_RUNG wire#w1
   // the same network as SCL:
   IF "PLC1_Stop_Active" OR "PLC1_Loi_Tong" THEN "V3341_Duong_Filter" := FALSE; END_IF;
END_REGION

REGION Network 60: Stop hoặc Lỗi tổng - reset Pump3264_Chuyen_Nhanh1
   RUNG wire#powerrail
      Contact( "PLC1_Stop_Active" )
      wire#w1
      R_Coil( "Pump3264_Chuyen_Nhanh1" )
   END_RUNG
   RUNG wire#powerrail
      Contact( "PLC1_Loi_Tong" )
   END_RUNG wire#w1
   // the same network as SCL:
   IF "PLC1_Stop_Active" OR "PLC1_Loi_Tong" THEN "Pump3264_Chuyen_Nhanh1" := FALSE; END_IF;
END_REGION

REGION Network 61: Stop hoặc Lỗi tổng - reset Pump3265_Chuyen_Nhanh2_Cmd
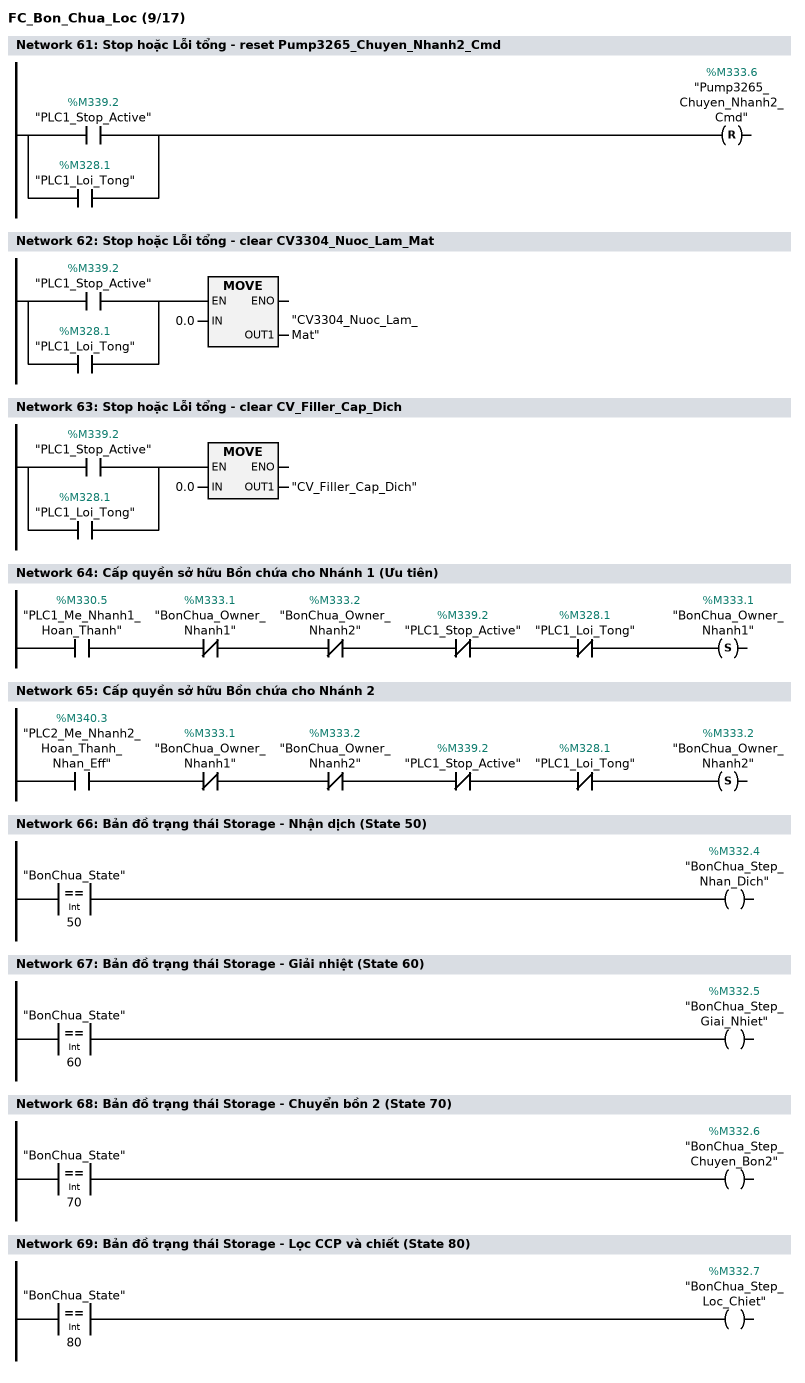
   RUNG wire#powerrail
      Contact( "PLC1_Stop_Active" )
      wire#w1
      R_Coil( "Pump3265_Chuyen_Nhanh2_Cmd" )
   END_RUNG
   RUNG wire#powerrail
      Contact( "PLC1_Loi_Tong" )
   END_RUNG wire#w1
   // the same network as SCL:
   IF "PLC1_Stop_Active" OR "PLC1_Loi_Tong" THEN "Pump3265_Chuyen_Nhanh2_Cmd" := FALSE; END_IF;
END_REGION

REGION Network 62: Stop hoặc Lỗi tổng - clear CV3304_Nuoc_Lam_Mat
   RUNG wire#powerrail
      Contact( "PLC1_Stop_Active" )
      wire#w1
      { S7_GenerateENO := "TRUE" } Move(in := 0.0, out1 => "CV3304_Nuoc_Lam_Mat")
   END_RUNG
   RUNG wire#powerrail
      Contact( "PLC1_Loi_Tong" )
   END_RUNG wire#w1
   // the same network as SCL:
   IF "PLC1_Stop_Active" OR "PLC1_Loi_Tong" THEN "CV3304_Nuoc_Lam_Mat" := 0.0; END_IF;
END_REGION

REGION Network 63: Stop hoặc Lỗi tổng - clear CV_Filler_Cap_Dich
   RUNG wire#powerrail
      Contact( "PLC1_Stop_Active" )
      wire#w1
      { S7_GenerateENO := "TRUE" } Move(in := 0.0, out1 => "CV_Filler_Cap_Dich")
   END_RUNG
   RUNG wire#powerrail
      Contact( "PLC1_Loi_Tong" )
   END_RUNG wire#w1
   // the same network as SCL:
   IF "PLC1_Stop_Active" OR "PLC1_Loi_Tong" THEN "CV_Filler_Cap_Dich" := 0.0; END_IF;
END_REGION

REGION Network 64: Cấp quyền sở hữu Bồn chứa cho Nhánh 1 (Ưu tiên)
   RUNG wire#powerrail
      Contact( "PLC1_Me_Nhanh1_Hoan_Thanh" )
      I_Contact( "BonChua_Owner_Nhanh1" )
      I_Contact( "BonChua_Owner_Nhanh2" )
      I_Contact( "PLC1_Stop_Active" )
      I_Contact( "PLC1_Loi_Tong" )
      S_Coil( "BonChua_Owner_Nhanh1" )
   END_RUNG
   // the same network as SCL:
   IF "PLC1_Me_Nhanh1_Hoan_Thanh" AND NOT "BonChua_Owner_Nhanh1" AND NOT "BonChua_Owner_Nhanh2" AND NOT "PLC1_Stop_Active" AND NOT "PLC1_Loi_Tong" THEN
       "BonChua_Owner_Nhanh1" := TRUE;
   END_IF;
END_REGION

REGION Network 65: Cấp quyền sở hữu Bồn chứa cho Nhánh 2
   RUNG wire#powerrail
      Contact( "PLC2_Me_Nhanh2_Hoan_Thanh_Nhan_Eff" )
      I_Contact( "BonChua_Owner_Nhanh1" )
      I_Contact( "BonChua_Owner_Nhanh2" )
      I_Contact( "PLC1_Stop_Active" )
      I_Contact( "PLC1_Loi_Tong" )
      S_Coil( "BonChua_Owner_Nhanh2" )
   END_RUNG
   // the same network as SCL:
   IF "PLC2_Me_Nhanh2_Hoan_Thanh_Nhan_Eff" AND NOT "BonChua_Owner_Nhanh1" AND NOT "BonChua_Owner_Nhanh2" AND NOT "PLC1_Stop_Active" AND NOT "PLC1_Loi_Tong" THEN
       "BonChua_Owner_Nhanh2" := TRUE;
   END_IF;
END_REGION

REGION Network 66: Bản đồ trạng thái Storage - Nhận dịch (State 50)
   RUNG wire#powerrail
      { S7_Templates := "SrcType := Int" } EQ_Contact(in1 := "BonChua_State", in2 := 50)
      Coil( "BonChua_Step_Nhan_Dich" )
   END_RUNG
   // the same network as SCL:
   "BonChua_Step_Nhan_Dich" := "BonChua_State" = 50;
END_REGION

REGION Network 67: Bản đồ trạng thái Storage - Giải nhiệt (State 60)
   RUNG wire#powerrail
      { S7_Templates := "SrcType := Int" } EQ_Contact(in1 := "BonChua_State", in2 := 60)
      Coil( "BonChua_Step_Giai_Nhiet" )
   END_RUNG
   // the same network as SCL:
   "BonChua_Step_Giai_Nhiet" := "BonChua_State" = 60;
END_REGION

REGION Network 68: Bản đồ trạng thái Storage - Chuyển bồn 2 (State 70)
   RUNG wire#powerrail
      { S7_Templates := "SrcType := Int" } EQ_Contact(in1 := "BonChua_State", in2 := 70)
      Coil( "BonChua_Step_Chuyen_Bon2" )
   END_RUNG
   // the same network as SCL:
   "BonChua_Step_Chuyen_Bon2" := "BonChua_State" = 70;
END_REGION

REGION Network 69: Bản đồ trạng thái Storage - Lọc CCP và chiết (State 80)
   RUNG wire#powerrail
      { S7_Templates := "SrcType := Int" } EQ_Contact(in1 := "BonChua_State", in2 := 80)
      Coil( "BonChua_Step_Loc_Chiet" )
   END_RUNG
   // the same network as SCL:
   "BonChua_Step_Loc_Chiet" := "BonChua_State" = 80;
END_REGION

REGION Network 70: Nhận mẻ từ Nhánh 1 hoặc Nhánh 2 thành công - Chuyển sang State 50
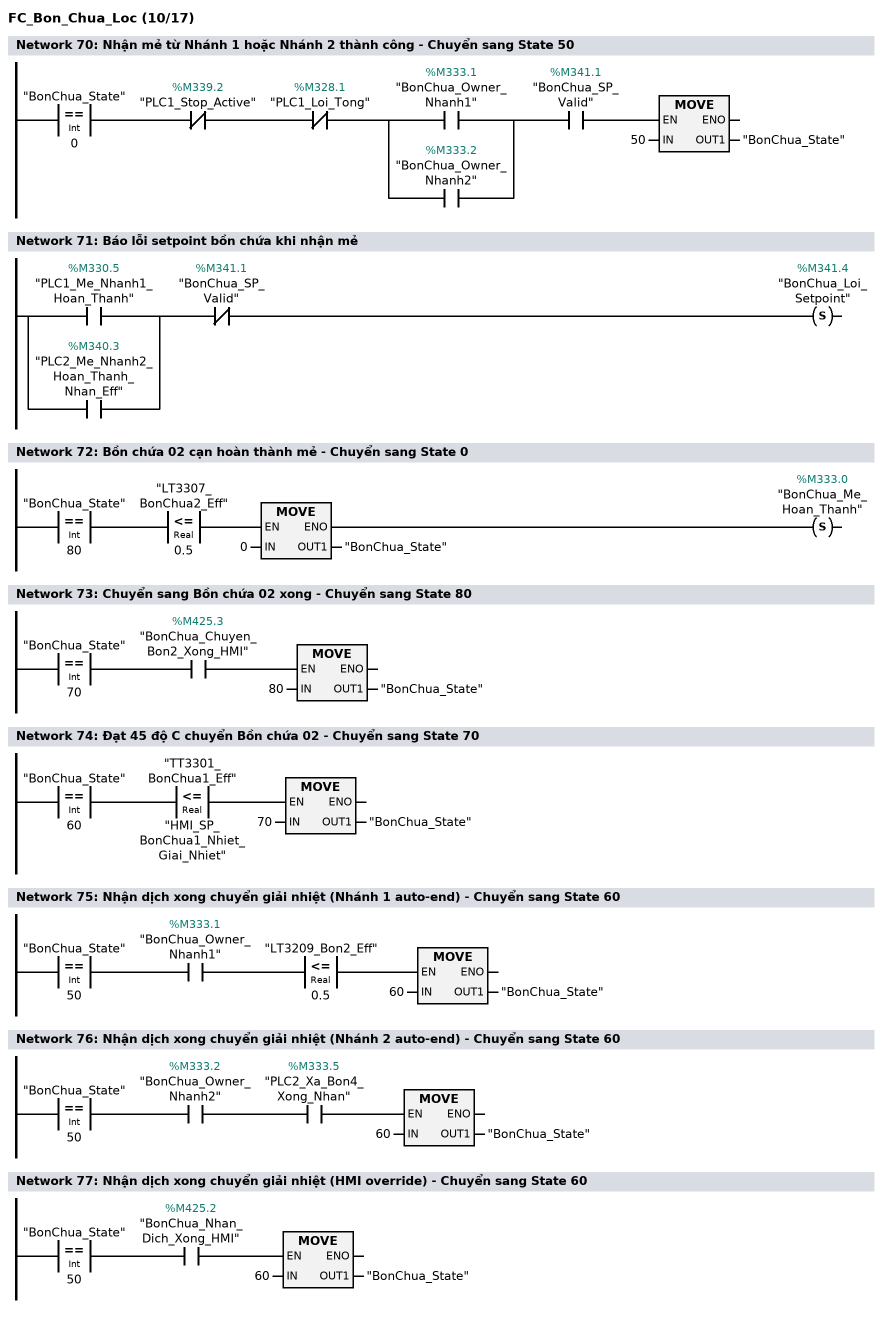
   RUNG wire#powerrail
      { S7_Templates := "SrcType := Int" } EQ_Contact(in1 := "BonChua_State", in2 := 0)
      I_Contact( "PLC1_Stop_Active" )
      I_Contact( "PLC1_Loi_Tong" )
      wire#w1
      Contact( "BonChua_Owner_Nhanh1" )
      wire#w2
      Contact( "BonChua_SP_Valid" )
      { S7_GenerateENO := "TRUE" } Move(in := 50, out1 => "BonChua_State")
   END_RUNG
   RUNG wire#w1
      Contact( "BonChua_Owner_Nhanh2" )
   END_RUNG wire#w2
   // the same network as SCL:
   IF ("BonChua_State" = 0) AND NOT "PLC1_Stop_Active" AND NOT "PLC1_Loi_Tong" AND ("BonChua_Owner_Nhanh1" OR "BonChua_Owner_Nhanh2") AND "BonChua_SP_Valid" THEN
       "BonChua_State" := 50;
   END_IF;
END_REGION

REGION Network 71: Báo lỗi setpoint bồn chứa khi nhận mẻ
   RUNG wire#powerrail
      Contact( "PLC1_Me_Nhanh1_Hoan_Thanh" )
      wire#w1
      I_Contact( "BonChua_SP_Valid" )
      S_Coil( "BonChua_Loi_Setpoint" )
   END_RUNG
   RUNG wire#powerrail
      Contact( "PLC2_Me_Nhanh2_Hoan_Thanh_Nhan_Eff" )
   END_RUNG wire#w1
   // the same network as SCL:
   IF ("PLC1_Me_Nhanh1_Hoan_Thanh" OR "PLC2_Me_Nhanh2_Hoan_Thanh_Nhan_Eff") AND NOT "BonChua_SP_Valid" THEN
       "BonChua_Loi_Setpoint" := TRUE;
   END_IF;
END_REGION

REGION Network 72: Bồn chứa 02 cạn hoàn thành mẻ - Chuyển sang State 0
   RUNG wire#powerrail
      { S7_Templates := "SrcType := Int" } EQ_Contact(in1 := "BonChua_State", in2 := 80)
      { S7_Templates := "SrcType := Real" } LE_Contact(in1 := "LT3307_BonChua2_Eff", in2 := 0.5)
      { S7_GenerateENO := "TRUE" } Move(in := 0, out1 => "BonChua_State")
      S_Coil( "BonChua_Me_Hoan_Thanh" )
   END_RUNG
   // the same network as SCL:
   // ENO of a box is taken as its EN; it also drops when the box reports an error
   #_w1 := ("BonChua_State" = 80) AND ("LT3307_BonChua2_Eff" <= 0.5);
   IF #_w1 THEN
       "BonChua_State" := 0;
       "BonChua_Me_Hoan_Thanh" := TRUE;
   END_IF;
END_REGION

REGION Network 73: Chuyển sang Bồn chứa 02 xong - Chuyển sang State 80
   RUNG wire#powerrail
      { S7_Templates := "SrcType := Int" } EQ_Contact(in1 := "BonChua_State", in2 := 70)
      Contact( "BonChua_Chuyen_Bon2_Xong_HMI" )
      { S7_GenerateENO := "TRUE" } Move(in := 80, out1 => "BonChua_State")
   END_RUNG
   // the same network as SCL:
   IF ("BonChua_State" = 70) AND "BonChua_Chuyen_Bon2_Xong_HMI" THEN "BonChua_State" := 80; END_IF;
END_REGION

REGION Network 74: Đạt 45 độ C chuyển Bồn chứa 02 - Chuyển sang State 70
   RUNG wire#powerrail
      { S7_Templates := "SrcType := Int" } EQ_Contact(in1 := "BonChua_State", in2 := 60)
      { S7_Templates := "SrcType := Real" } LE_Contact(in1 := "TT3301_BonChua1_Eff", in2 := "HMI_SP_BonChua1_Nhiet_Giai_Nhiet")
      { S7_GenerateENO := "TRUE" } Move(in := 70, out1 => "BonChua_State")
   END_RUNG
   // the same network as SCL:
   IF ("BonChua_State" = 60) AND ("TT3301_BonChua1_Eff" <= "HMI_SP_BonChua1_Nhiet_Giai_Nhiet") THEN
       "BonChua_State" := 70;
   END_IF;
END_REGION

REGION Network 75: Nhận dịch xong chuyển giải nhiệt (Nhánh 1 auto-end) - Chuyển sang State 60
   RUNG wire#powerrail
      { S7_Templates := "SrcType := Int" } EQ_Contact(in1 := "BonChua_State", in2 := 50)
      Contact( "BonChua_Owner_Nhanh1" )
      { S7_Templates := "SrcType := Real" } LE_Contact(in1 := "LT3209_Bon2_Eff", in2 := 0.5)
      { S7_GenerateENO := "TRUE" } Move(in := 60, out1 => "BonChua_State")
   END_RUNG
   // the same network as SCL:
   IF ("BonChua_State" = 50) AND "BonChua_Owner_Nhanh1" AND ("LT3209_Bon2_Eff" <= 0.5) THEN
       "BonChua_State" := 60;
   END_IF;
END_REGION

REGION Network 76: Nhận dịch xong chuyển giải nhiệt (Nhánh 2 auto-end) - Chuyển sang State 60
   RUNG wire#powerrail
      { S7_Templates := "SrcType := Int" } EQ_Contact(in1 := "BonChua_State", in2 := 50)
      Contact( "BonChua_Owner_Nhanh2" )
      Contact( "PLC2_Xa_Bon4_Xong_Nhan" )
      { S7_GenerateENO := "TRUE" } Move(in := 60, out1 => "BonChua_State")
   END_RUNG
   // the same network as SCL:
   IF ("BonChua_State" = 50) AND "BonChua_Owner_Nhanh2" AND "PLC2_Xa_Bon4_Xong_Nhan" THEN
       "BonChua_State" := 60;
   END_IF;
END_REGION

REGION Network 77: Nhận dịch xong chuyển giải nhiệt (HMI override) - Chuyển sang State 60
   RUNG wire#powerrail
      { S7_Templates := "SrcType := Int" } EQ_Contact(in1 := "BonChua_State", in2 := 50)
      Contact( "BonChua_Nhan_Dich_Xong_HMI" )
      { S7_GenerateENO := "TRUE" } Move(in := 60, out1 => "BonChua_State")
   END_RUNG
   // the same network as SCL:
   IF ("BonChua_State" = 50) AND "BonChua_Nhan_Dich_Xong_HMI" THEN "BonChua_State" := 60; END_IF;
END_REGION

REGION Network 78: Reset cờ hoàn thành mẻ khi bắt đầu nhận dịch mới
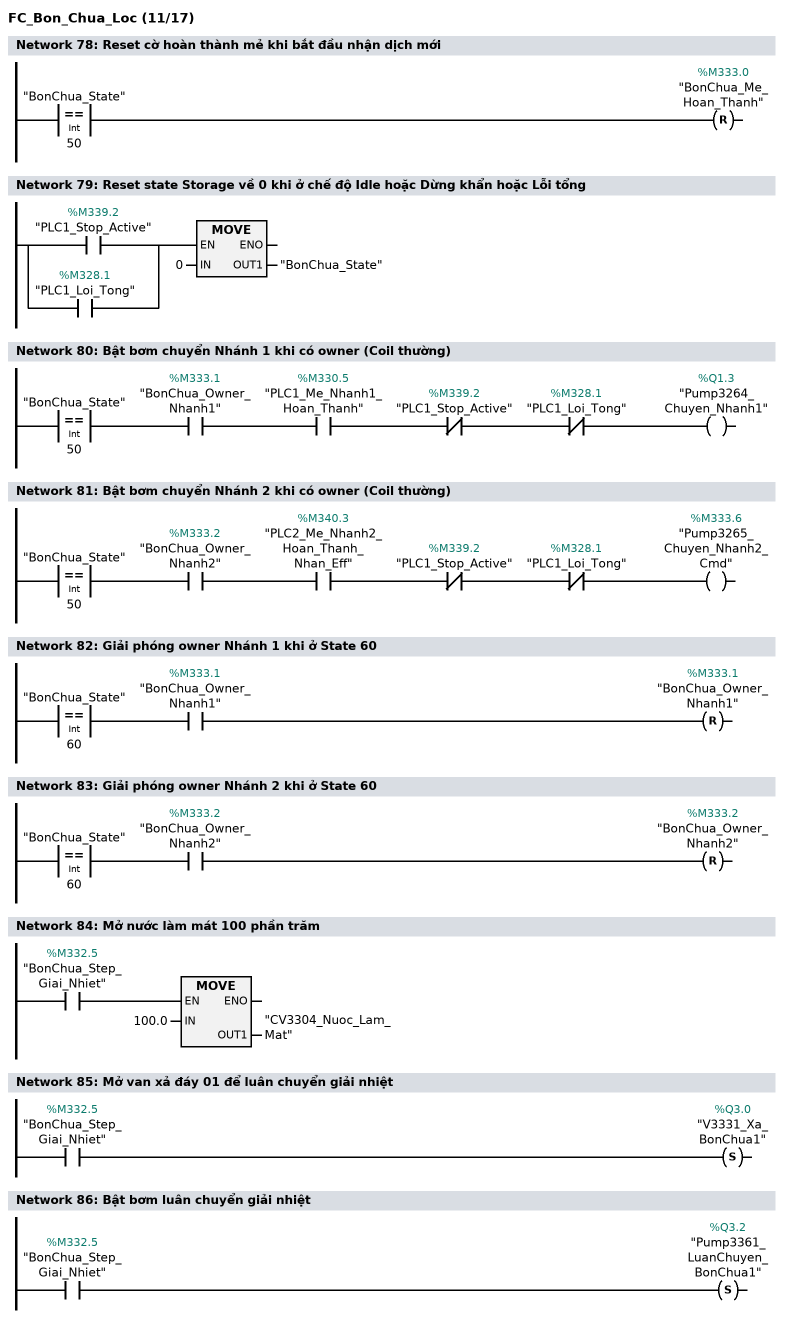
   RUNG wire#powerrail
      { S7_Templates := "SrcType := Int" } EQ_Contact(in1 := "BonChua_State", in2 := 50)
      R_Coil( "BonChua_Me_Hoan_Thanh" )
   END_RUNG
   // the same network as SCL:
   IF "BonChua_State" = 50 THEN "BonChua_Me_Hoan_Thanh" := FALSE; END_IF;
END_REGION

REGION Network 79: Reset state Storage về 0 khi ở chế độ Idle hoặc Dừng khẩn hoặc Lỗi tổng
   RUNG wire#powerrail
      Contact( "PLC1_Stop_Active" )
      wire#w1
      { S7_GenerateENO := "TRUE" } Move(in := 0, out1 => "BonChua_State")
   END_RUNG
   RUNG wire#powerrail
      Contact( "PLC1_Loi_Tong" )
   END_RUNG wire#w1
   // the same network as SCL:
   IF "PLC1_Stop_Active" OR "PLC1_Loi_Tong" THEN "BonChua_State" := 0; END_IF;
END_REGION

REGION Network 80: Bật bơm chuyển Nhánh 1 khi có owner (Coil thường)
   RUNG wire#powerrail
      { S7_Templates := "SrcType := Int" } EQ_Contact(in1 := "BonChua_State", in2 := 50)
      Contact( "BonChua_Owner_Nhanh1" )
      Contact( "PLC1_Me_Nhanh1_Hoan_Thanh" )
      I_Contact( "PLC1_Stop_Active" )
      I_Contact( "PLC1_Loi_Tong" )
      Coil( "Pump3264_Chuyen_Nhanh1" )
   END_RUNG
   // the same network as SCL:
   "Pump3264_Chuyen_Nhanh1" := ("BonChua_State" = 50) AND "BonChua_Owner_Nhanh1" AND "PLC1_Me_Nhanh1_Hoan_Thanh" AND NOT "PLC1_Stop_Active" AND NOT "PLC1_Loi_Tong";
END_REGION

REGION Network 81: Bật bơm chuyển Nhánh 2 khi có owner (Coil thường)
   RUNG wire#powerrail
      { S7_Templates := "SrcType := Int" } EQ_Contact(in1 := "BonChua_State", in2 := 50)
      Contact( "BonChua_Owner_Nhanh2" )
      Contact( "PLC2_Me_Nhanh2_Hoan_Thanh_Nhan_Eff" )
      I_Contact( "PLC1_Stop_Active" )
      I_Contact( "PLC1_Loi_Tong" )
      Coil( "Pump3265_Chuyen_Nhanh2_Cmd" )
   END_RUNG
   // the same network as SCL:
   "Pump3265_Chuyen_Nhanh2_Cmd" := ("BonChua_State" = 50) AND "BonChua_Owner_Nhanh2" AND "PLC2_Me_Nhanh2_Hoan_Thanh_Nhan_Eff" AND NOT "PLC1_Stop_Active" AND NOT "PLC1_Loi_Tong";
END_REGION

REGION Network 82: Giải phóng owner Nhánh 1 khi ở State 60
   RUNG wire#powerrail
      { S7_Templates := "SrcType := Int" } EQ_Contact(in1 := "BonChua_State", in2 := 60)
      Contact( "BonChua_Owner_Nhanh1" )
      R_Coil( "BonChua_Owner_Nhanh1" )
   END_RUNG
   // the same network as SCL:
   IF ("BonChua_State" = 60) AND "BonChua_Owner_Nhanh1" THEN "BonChua_Owner_Nhanh1" := FALSE; END_IF;
END_REGION

REGION Network 83: Giải phóng owner Nhánh 2 khi ở State 60
   RUNG wire#powerrail
      { S7_Templates := "SrcType := Int" } EQ_Contact(in1 := "BonChua_State", in2 := 60)
      Contact( "BonChua_Owner_Nhanh2" )
      R_Coil( "BonChua_Owner_Nhanh2" )
   END_RUNG
   // the same network as SCL:
   IF ("BonChua_State" = 60) AND "BonChua_Owner_Nhanh2" THEN "BonChua_Owner_Nhanh2" := FALSE; END_IF;
END_REGION

REGION Network 84: Mở nước làm mát 100 phần trăm
   RUNG wire#powerrail
      Contact( "BonChua_Step_Giai_Nhiet" )
      { S7_GenerateENO := "TRUE" } Move(in := 100.0, out1 => "CV3304_Nuoc_Lam_Mat")
   END_RUNG
   // the same network as SCL:
   IF "BonChua_Step_Giai_Nhiet" THEN "CV3304_Nuoc_Lam_Mat" := 100.0; END_IF;
END_REGION

REGION Network 85: Mở van xả đáy 01 để luân chuyển giải nhiệt
   RUNG wire#powerrail
      Contact( "BonChua_Step_Giai_Nhiet" )
      S_Coil( "V3331_Xa_BonChua1" )
   END_RUNG
   // the same network as SCL:
   IF "BonChua_Step_Giai_Nhiet" THEN "V3331_Xa_BonChua1" := TRUE; END_IF;
END_REGION

REGION Network 86: Bật bơm luân chuyển giải nhiệt
   RUNG wire#powerrail
      Contact( "BonChua_Step_Giai_Nhiet" )
      S_Coil( "Pump3361_LuanChuyen_BonChua1" )
   END_RUNG
   // the same network as SCL:
   IF "BonChua_Step_Giai_Nhiet" THEN "Pump3361_LuanChuyen_BonChua1" := TRUE; END_IF;
END_REGION

REGION Network 87: Đóng van hơi giải nhiệt
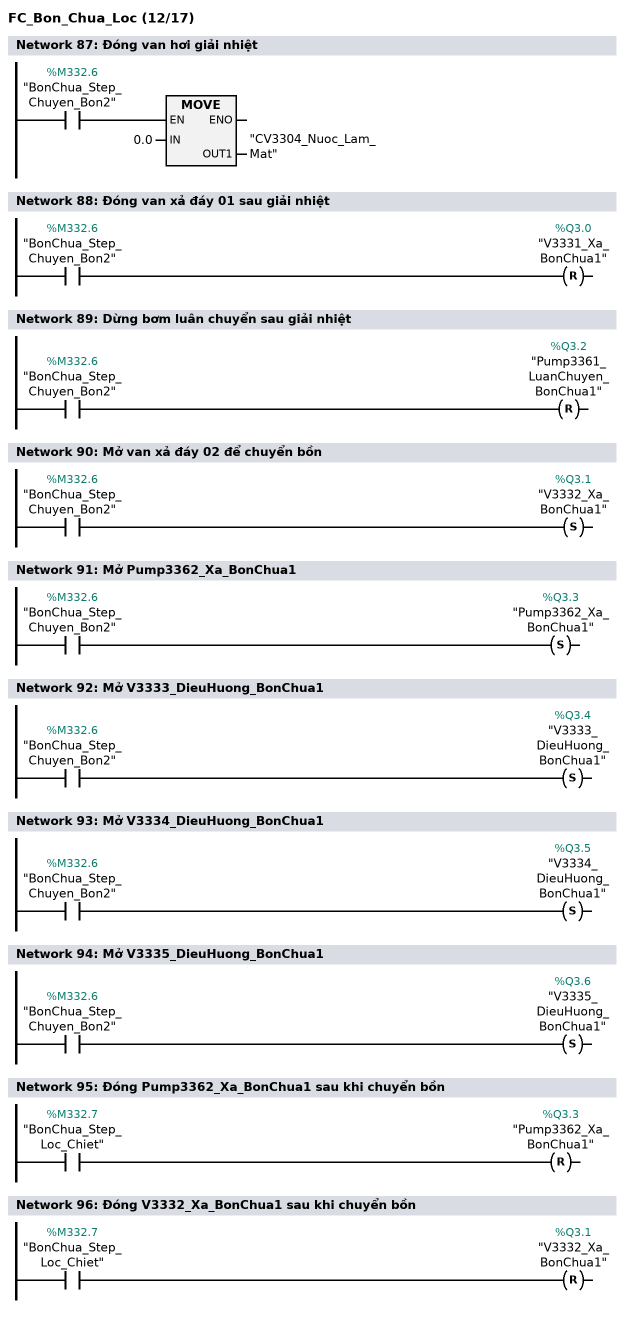
   RUNG wire#powerrail
      Contact( "BonChua_Step_Chuyen_Bon2" )
      { S7_GenerateENO := "TRUE" } Move(in := 0.0, out1 => "CV3304_Nuoc_Lam_Mat")
   END_RUNG
   // the same network as SCL:
   IF "BonChua_Step_Chuyen_Bon2" THEN "CV3304_Nuoc_Lam_Mat" := 0.0; END_IF;
END_REGION

REGION Network 88: Đóng van xả đáy 01 sau giải nhiệt
   RUNG wire#powerrail
      Contact( "BonChua_Step_Chuyen_Bon2" )
      R_Coil( "V3331_Xa_BonChua1" )
   END_RUNG
   // the same network as SCL:
   IF "BonChua_Step_Chuyen_Bon2" THEN "V3331_Xa_BonChua1" := FALSE; END_IF;
END_REGION

REGION Network 89: Dừng bơm luân chuyển sau giải nhiệt
   RUNG wire#powerrail
      Contact( "BonChua_Step_Chuyen_Bon2" )
      R_Coil( "Pump3361_LuanChuyen_BonChua1" )
   END_RUNG
   // the same network as SCL:
   IF "BonChua_Step_Chuyen_Bon2" THEN "Pump3361_LuanChuyen_BonChua1" := FALSE; END_IF;
END_REGION

REGION Network 90: Mở van xả đáy 02 để chuyển bồn
   RUNG wire#powerrail
      Contact( "BonChua_Step_Chuyen_Bon2" )
      S_Coil( "V3332_Xa_BonChua1" )
   END_RUNG
   // the same network as SCL:
   IF "BonChua_Step_Chuyen_Bon2" THEN "V3332_Xa_BonChua1" := TRUE; END_IF;
END_REGION

REGION Network 91: Mở Pump3362_Xa_BonChua1
   RUNG wire#powerrail
      Contact( "BonChua_Step_Chuyen_Bon2" )
      S_Coil( "Pump3362_Xa_BonChua1" )
   END_RUNG
   // the same network as SCL:
   IF "BonChua_Step_Chuyen_Bon2" THEN "Pump3362_Xa_BonChua1" := TRUE; END_IF;
END_REGION

REGION Network 92: Mở V3333_DieuHuong_BonChua1
   RUNG wire#powerrail
      Contact( "BonChua_Step_Chuyen_Bon2" )
      S_Coil( "V3333_DieuHuong_BonChua1" )
   END_RUNG
   // the same network as SCL:
   IF "BonChua_Step_Chuyen_Bon2" THEN "V3333_DieuHuong_BonChua1" := TRUE; END_IF;
END_REGION

REGION Network 93: Mở V3334_DieuHuong_BonChua1
   RUNG wire#powerrail
      Contact( "BonChua_Step_Chuyen_Bon2" )
      S_Coil( "V3334_DieuHuong_BonChua1" )
   END_RUNG
   // the same network as SCL:
   IF "BonChua_Step_Chuyen_Bon2" THEN "V3334_DieuHuong_BonChua1" := TRUE; END_IF;
END_REGION

REGION Network 94: Mở V3335_DieuHuong_BonChua1
   RUNG wire#powerrail
      Contact( "BonChua_Step_Chuyen_Bon2" )
      S_Coil( "V3335_DieuHuong_BonChua1" )
   END_RUNG
   // the same network as SCL:
   IF "BonChua_Step_Chuyen_Bon2" THEN "V3335_DieuHuong_BonChua1" := TRUE; END_IF;
END_REGION

REGION Network 95: Đóng Pump3362_Xa_BonChua1 sau khi chuyển bồn
   RUNG wire#powerrail
      Contact( "BonChua_Step_Loc_Chiet" )
      R_Coil( "Pump3362_Xa_BonChua1" )
   END_RUNG
   // the same network as SCL:
   IF "BonChua_Step_Loc_Chiet" THEN "Pump3362_Xa_BonChua1" := FALSE; END_IF;
END_REGION

REGION Network 96: Đóng V3332_Xa_BonChua1 sau khi chuyển bồn
   RUNG wire#powerrail
      Contact( "BonChua_Step_Loc_Chiet" )
      R_Coil( "V3332_Xa_BonChua1" )
   END_RUNG
   // the same network as SCL:
   IF "BonChua_Step_Loc_Chiet" THEN "V3332_Xa_BonChua1" := FALSE; END_IF;
END_REGION

REGION Network 97: Đóng V3333_DieuHuong_BonChua1 sau khi chuyển bồn
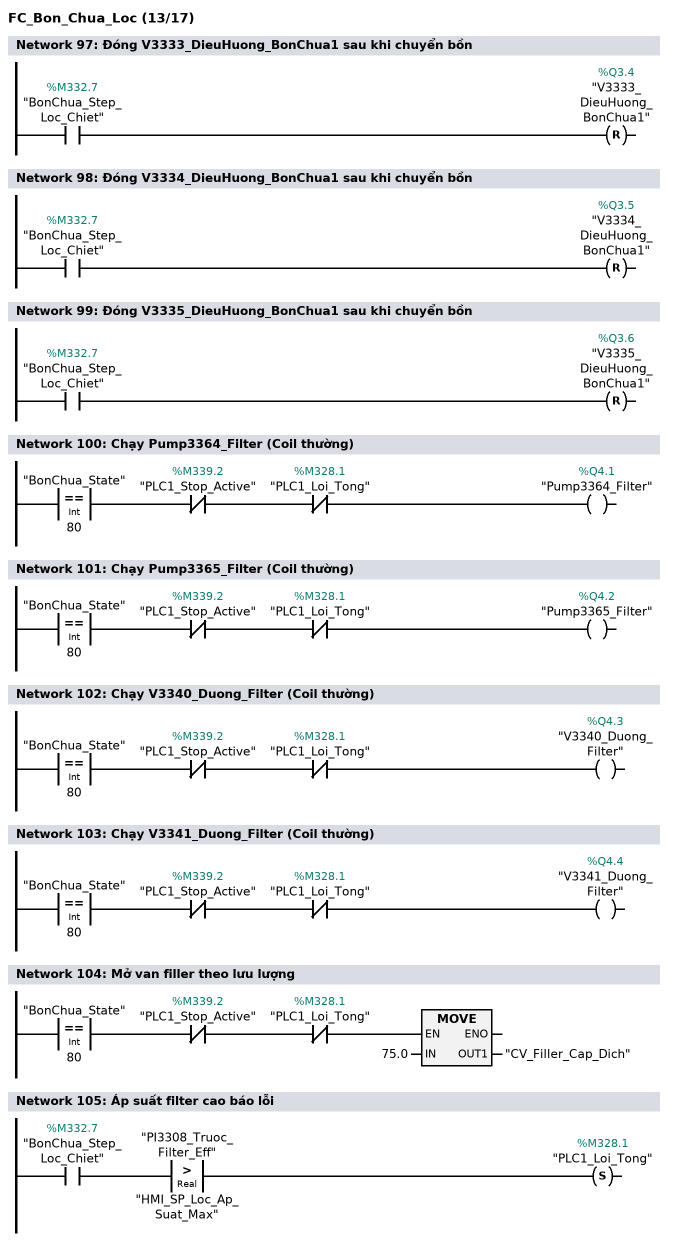
   RUNG wire#powerrail
      Contact( "BonChua_Step_Loc_Chiet" )
      R_Coil( "V3333_DieuHuong_BonChua1" )
   END_RUNG
   // the same network as SCL:
   IF "BonChua_Step_Loc_Chiet" THEN "V3333_DieuHuong_BonChua1" := FALSE; END_IF;
END_REGION

REGION Network 98: Đóng V3334_DieuHuong_BonChua1 sau khi chuyển bồn
   RUNG wire#powerrail
      Contact( "BonChua_Step_Loc_Chiet" )
      R_Coil( "V3334_DieuHuong_BonChua1" )
   END_RUNG
   // the same network as SCL:
   IF "BonChua_Step_Loc_Chiet" THEN "V3334_DieuHuong_BonChua1" := FALSE; END_IF;
END_REGION

REGION Network 99: Đóng V3335_DieuHuong_BonChua1 sau khi chuyển bồn
   RUNG wire#powerrail
      Contact( "BonChua_Step_Loc_Chiet" )
      R_Coil( "V3335_DieuHuong_BonChua1" )
   END_RUNG
   // the same network as SCL:
   IF "BonChua_Step_Loc_Chiet" THEN "V3335_DieuHuong_BonChua1" := FALSE; END_IF;
END_REGION

REGION Network 100: Chạy Pump3364_Filter (Coil thường)
   RUNG wire#powerrail
      { S7_Templates := "SrcType := Int" } EQ_Contact(in1 := "BonChua_State", in2 := 80)
      I_Contact( "PLC1_Stop_Active" )
      I_Contact( "PLC1_Loi_Tong" )
      Coil( "Pump3364_Filter" )
   END_RUNG
   // the same network as SCL:
   "Pump3364_Filter" := ("BonChua_State" = 80) AND NOT "PLC1_Stop_Active" AND NOT "PLC1_Loi_Tong";
END_REGION

REGION Network 101: Chạy Pump3365_Filter (Coil thường)
   RUNG wire#powerrail
      { S7_Templates := "SrcType := Int" } EQ_Contact(in1 := "BonChua_State", in2 := 80)
      I_Contact( "PLC1_Stop_Active" )
      I_Contact( "PLC1_Loi_Tong" )
      Coil( "Pump3365_Filter" )
   END_RUNG
   // the same network as SCL:
   "Pump3365_Filter" := ("BonChua_State" = 80) AND NOT "PLC1_Stop_Active" AND NOT "PLC1_Loi_Tong";
END_REGION

REGION Network 102: Chạy V3340_Duong_Filter (Coil thường)
   RUNG wire#powerrail
      { S7_Templates := "SrcType := Int" } EQ_Contact(in1 := "BonChua_State", in2 := 80)
      I_Contact( "PLC1_Stop_Active" )
      I_Contact( "PLC1_Loi_Tong" )
      Coil( "V3340_Duong_Filter" )
   END_RUNG
   // the same network as SCL:
   "V3340_Duong_Filter" := ("BonChua_State" = 80) AND NOT "PLC1_Stop_Active" AND NOT "PLC1_Loi_Tong";
END_REGION

REGION Network 103: Chạy V3341_Duong_Filter (Coil thường)
   RUNG wire#powerrail
      { S7_Templates := "SrcType := Int" } EQ_Contact(in1 := "BonChua_State", in2 := 80)
      I_Contact( "PLC1_Stop_Active" )
      I_Contact( "PLC1_Loi_Tong" )
      Coil( "V3341_Duong_Filter" )
   END_RUNG
   // the same network as SCL:
   "V3341_Duong_Filter" := ("BonChua_State" = 80) AND NOT "PLC1_Stop_Active" AND NOT "PLC1_Loi_Tong";
END_REGION

REGION Network 104: Mở van filler theo lưu lượng
   RUNG wire#powerrail
      { S7_Templates := "SrcType := Int" } EQ_Contact(in1 := "BonChua_State", in2 := 80)
      I_Contact( "PLC1_Stop_Active" )
      I_Contact( "PLC1_Loi_Tong" )
      { S7_GenerateENO := "TRUE" } Move(in := 75.0, out1 => "CV_Filler_Cap_Dich")
   END_RUNG
   // the same network as SCL:
   IF ("BonChua_State" = 80) AND NOT "PLC1_Stop_Active" AND NOT "PLC1_Loi_Tong" THEN
       "CV_Filler_Cap_Dich" := 75.0;
   END_IF;
END_REGION

REGION Network 105: Áp suất filter cao báo lỗi
   RUNG wire#powerrail
      Contact( "BonChua_Step_Loc_Chiet" )
      { S7_Templates := "SrcType := Real" } GT_Contact(in1 := "PI3308_Truoc_Filter_Eff", in2 := "HMI_SP_Loc_Ap_Suat_Max")
      S_Coil( "PLC1_Loi_Tong" )
   END_RUNG
   // the same network as SCL:
   IF "BonChua_Step_Loc_Chiet" AND ("PI3308_Truoc_Filter_Eff" > "HMI_SP_Loc_Ap_Suat_Max") THEN
       "PLC1_Loi_Tong" := TRUE;
   END_IF;
END_REGION

REGION Network 106: Reset CV nước làm mát khi không giải nhiệt
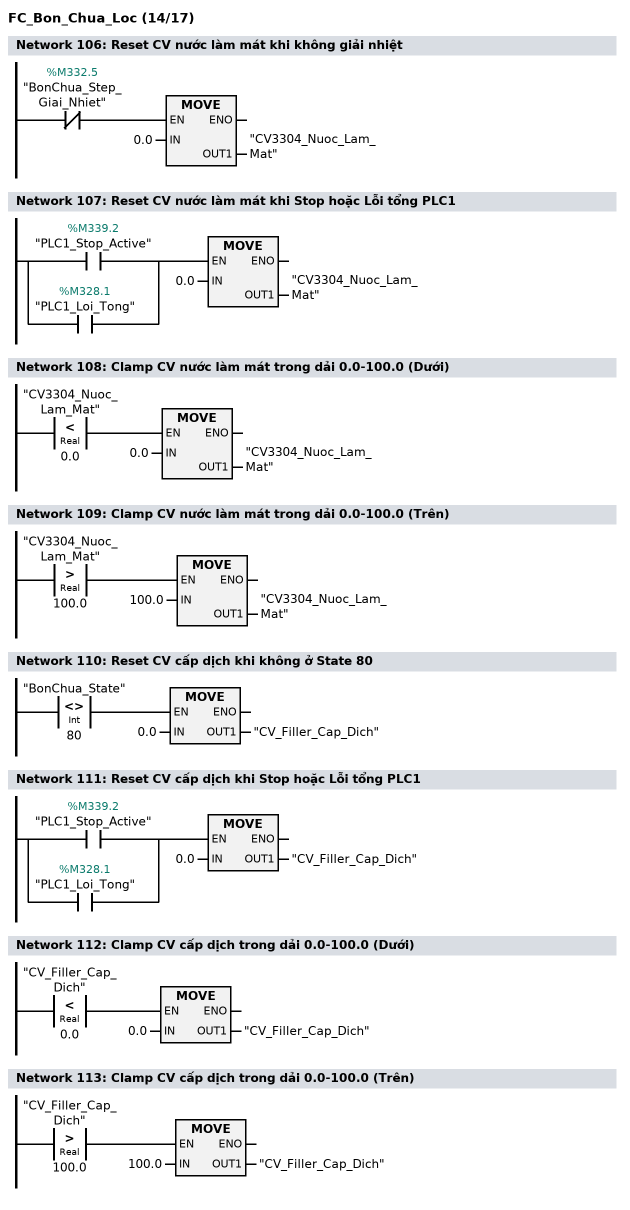
   RUNG wire#powerrail
      I_Contact( "BonChua_Step_Giai_Nhiet" )
      { S7_GenerateENO := "TRUE" } Move(in := 0.0, out1 => "CV3304_Nuoc_Lam_Mat")
   END_RUNG
   // the same network as SCL:
   IF NOT "BonChua_Step_Giai_Nhiet" THEN "CV3304_Nuoc_Lam_Mat" := 0.0; END_IF;
END_REGION

REGION Network 107: Reset CV nước làm mát khi Stop hoặc Lỗi tổng PLC1
   RUNG wire#powerrail
      Contact( "PLC1_Stop_Active" )
      wire#w1
      { S7_GenerateENO := "TRUE" } Move(in := 0.0, out1 => "CV3304_Nuoc_Lam_Mat")
   END_RUNG
   RUNG wire#powerrail
      Contact( "PLC1_Loi_Tong" )
   END_RUNG wire#w1
   // the same network as SCL:
   IF "PLC1_Stop_Active" OR "PLC1_Loi_Tong" THEN "CV3304_Nuoc_Lam_Mat" := 0.0; END_IF;
END_REGION

REGION Network 108: Clamp CV nước làm mát trong dải 0.0-100.0 (Dưới)
   RUNG wire#powerrail
      { S7_Templates := "SrcType := Real" } LT_Contact(in1 := "CV3304_Nuoc_Lam_Mat", in2 := 0.0)
      { S7_GenerateENO := "TRUE" } Move(in := 0.0, out1 => "CV3304_Nuoc_Lam_Mat")
   END_RUNG
   // the same network as SCL:
   IF "CV3304_Nuoc_Lam_Mat" < 0.0 THEN "CV3304_Nuoc_Lam_Mat" := 0.0; END_IF;
END_REGION

REGION Network 109: Clamp CV nước làm mát trong dải 0.0-100.0 (Trên)
   RUNG wire#powerrail
      { S7_Templates := "SrcType := Real" } GT_Contact(in1 := "CV3304_Nuoc_Lam_Mat", in2 := 100.0)
      { S7_GenerateENO := "TRUE" } Move(in := 100.0, out1 => "CV3304_Nuoc_Lam_Mat")
   END_RUNG
   // the same network as SCL:
   IF "CV3304_Nuoc_Lam_Mat" > 100.0 THEN "CV3304_Nuoc_Lam_Mat" := 100.0; END_IF;
END_REGION

REGION Network 110: Reset CV cấp dịch khi không ở State 80
   RUNG wire#powerrail
      { S7_Templates := "SrcType := Int" } NE_Contact(in1 := "BonChua_State", in2 := 80)
      { S7_GenerateENO := "TRUE" } Move(in := 0.0, out1 => "CV_Filler_Cap_Dich")
   END_RUNG
   // the same network as SCL:
   IF "BonChua_State" <> 80 THEN "CV_Filler_Cap_Dich" := 0.0; END_IF;
END_REGION

REGION Network 111: Reset CV cấp dịch khi Stop hoặc Lỗi tổng PLC1
   RUNG wire#powerrail
      Contact( "PLC1_Stop_Active" )
      wire#w1
      { S7_GenerateENO := "TRUE" } Move(in := 0.0, out1 => "CV_Filler_Cap_Dich")
   END_RUNG
   RUNG wire#powerrail
      Contact( "PLC1_Loi_Tong" )
   END_RUNG wire#w1
   // the same network as SCL:
   IF "PLC1_Stop_Active" OR "PLC1_Loi_Tong" THEN "CV_Filler_Cap_Dich" := 0.0; END_IF;
END_REGION

REGION Network 112: Clamp CV cấp dịch trong dải 0.0-100.0 (Dưới)
   RUNG wire#powerrail
      { S7_Templates := "SrcType := Real" } LT_Contact(in1 := "CV_Filler_Cap_Dich", in2 := 0.0)
      { S7_GenerateENO := "TRUE" } Move(in := 0.0, out1 => "CV_Filler_Cap_Dich")
   END_RUNG
   // the same network as SCL:
   IF "CV_Filler_Cap_Dich" < 0.0 THEN "CV_Filler_Cap_Dich" := 0.0; END_IF;
END_REGION

REGION Network 113: Clamp CV cấp dịch trong dải 0.0-100.0 (Trên)
   RUNG wire#powerrail
      { S7_Templates := "SrcType := Real" } GT_Contact(in1 := "CV_Filler_Cap_Dich", in2 := 100.0)
      { S7_GenerateENO := "TRUE" } Move(in := 100.0, out1 => "CV_Filler_Cap_Dich")
   END_RUNG
   // the same network as SCL:
   IF "CV_Filler_Cap_Dich" > 100.0 THEN "CV_Filler_Cap_Dich" := 100.0; END_IF;
END_REGION

REGION Network 114: Reset BonChua_Step_Nhan_Dich khi Stop hoặc Lỗi tổng PLC1
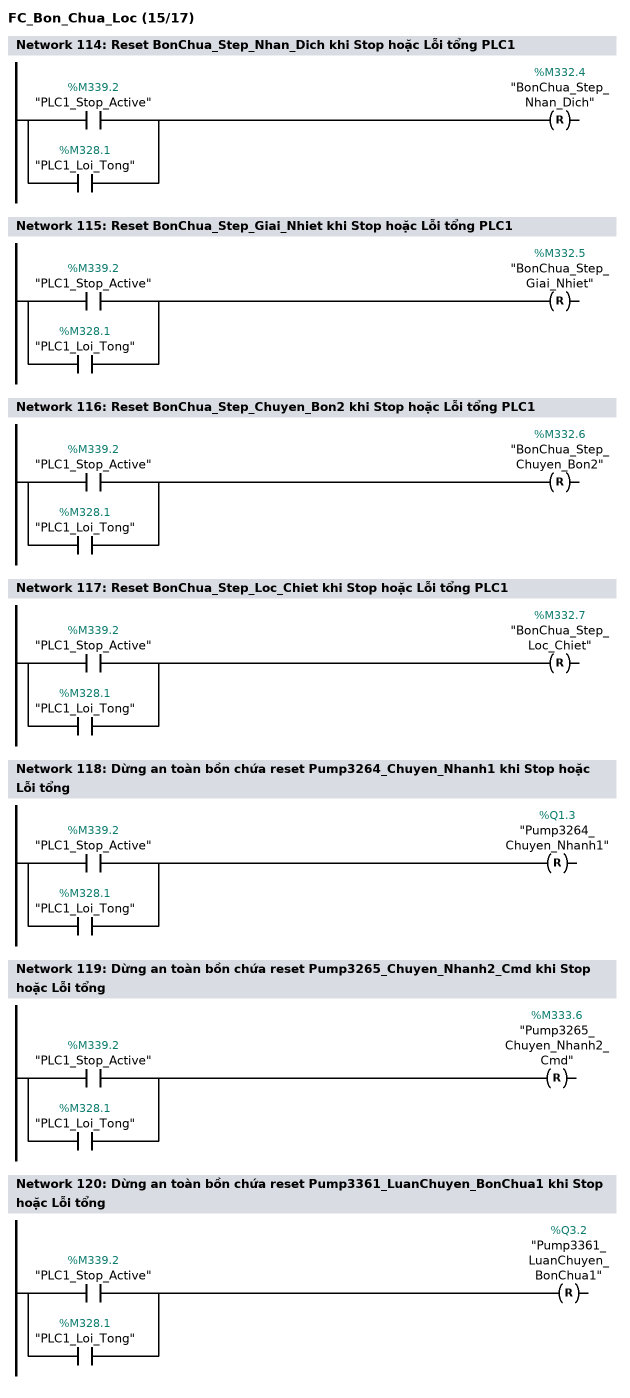
   RUNG wire#powerrail
      Contact( "PLC1_Stop_Active" )
      wire#w1
      R_Coil( "BonChua_Step_Nhan_Dich" )
   END_RUNG
   RUNG wire#powerrail
      Contact( "PLC1_Loi_Tong" )
   END_RUNG wire#w1
   // the same network as SCL:
   IF "PLC1_Stop_Active" OR "PLC1_Loi_Tong" THEN "BonChua_Step_Nhan_Dich" := FALSE; END_IF;
END_REGION

REGION Network 115: Reset BonChua_Step_Giai_Nhiet khi Stop hoặc Lỗi tổng PLC1
   RUNG wire#powerrail
      Contact( "PLC1_Stop_Active" )
      wire#w1
      R_Coil( "BonChua_Step_Giai_Nhiet" )
   END_RUNG
   RUNG wire#powerrail
      Contact( "PLC1_Loi_Tong" )
   END_RUNG wire#w1
   // the same network as SCL:
   IF "PLC1_Stop_Active" OR "PLC1_Loi_Tong" THEN "BonChua_Step_Giai_Nhiet" := FALSE; END_IF;
END_REGION

REGION Network 116: Reset BonChua_Step_Chuyen_Bon2 khi Stop hoặc Lỗi tổng PLC1
   RUNG wire#powerrail
      Contact( "PLC1_Stop_Active" )
      wire#w1
      R_Coil( "BonChua_Step_Chuyen_Bon2" )
   END_RUNG
   RUNG wire#powerrail
      Contact( "PLC1_Loi_Tong" )
   END_RUNG wire#w1
   // the same network as SCL:
   IF "PLC1_Stop_Active" OR "PLC1_Loi_Tong" THEN "BonChua_Step_Chuyen_Bon2" := FALSE; END_IF;
END_REGION

REGION Network 117: Reset BonChua_Step_Loc_Chiet khi Stop hoặc Lỗi tổng PLC1
   RUNG wire#powerrail
      Contact( "PLC1_Stop_Active" )
      wire#w1
      R_Coil( "BonChua_Step_Loc_Chiet" )
   END_RUNG
   RUNG wire#powerrail
      Contact( "PLC1_Loi_Tong" )
   END_RUNG wire#w1
   // the same network as SCL:
   IF "PLC1_Stop_Active" OR "PLC1_Loi_Tong" THEN "BonChua_Step_Loc_Chiet" := FALSE; END_IF;
END_REGION

REGION Network 118: Dừng an toàn bồn chứa reset Pump3264_Chuyen_Nhanh1 khi Stop hoặc Lỗi tổng
   RUNG wire#powerrail
      Contact( "PLC1_Stop_Active" )
      wire#w1
      R_Coil( "Pump3264_Chuyen_Nhanh1" )
   END_RUNG
   RUNG wire#powerrail
      Contact( "PLC1_Loi_Tong" )
   END_RUNG wire#w1
   // the same network as SCL:
   IF "PLC1_Stop_Active" OR "PLC1_Loi_Tong" THEN "Pump3264_Chuyen_Nhanh1" := FALSE; END_IF;
END_REGION

REGION Network 119: Dừng an toàn bồn chứa reset Pump3265_Chuyen_Nhanh2_Cmd khi Stop hoặc Lỗi tổng
   RUNG wire#powerrail
      Contact( "PLC1_Stop_Active" )
      wire#w1
      R_Coil( "Pump3265_Chuyen_Nhanh2_Cmd" )
   END_RUNG
   RUNG wire#powerrail
      Contact( "PLC1_Loi_Tong" )
   END_RUNG wire#w1
   // the same network as SCL:
   IF "PLC1_Stop_Active" OR "PLC1_Loi_Tong" THEN "Pump3265_Chuyen_Nhanh2_Cmd" := FALSE; END_IF;
END_REGION

REGION Network 120: Dừng an toàn bồn chứa reset Pump3361_LuanChuyen_BonChua1 khi Stop hoặc Lỗi tổng
   RUNG wire#powerrail
      Contact( "PLC1_Stop_Active" )
      wire#w1
      R_Coil( "Pump3361_LuanChuyen_BonChua1" )
   END_RUNG
   RUNG wire#powerrail
      Contact( "PLC1_Loi_Tong" )
   END_RUNG wire#w1
   // the same network as SCL:
   IF "PLC1_Stop_Active" OR "PLC1_Loi_Tong" THEN "Pump3361_LuanChuyen_BonChua1" := FALSE; END_IF;
END_REGION

REGION Network 121: Dừng an toàn bồn chứa reset Pump3362_Xa_BonChua1 khi Stop hoặc Lỗi tổng
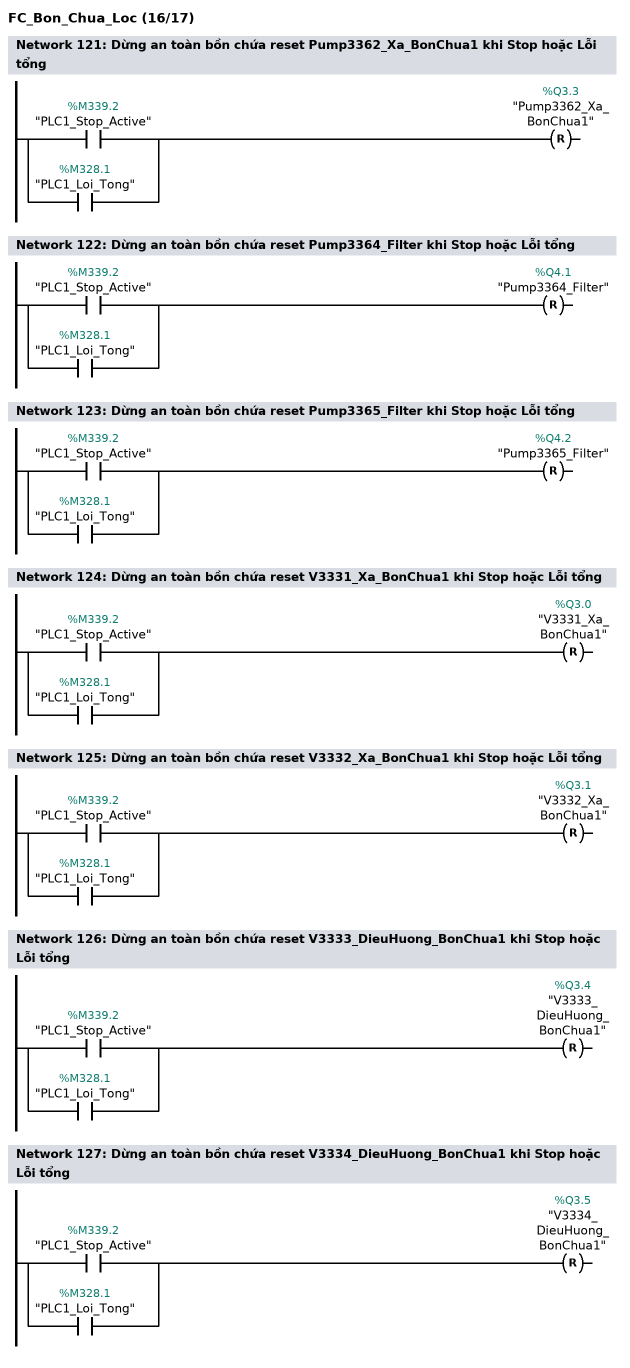
   RUNG wire#powerrail
      Contact( "PLC1_Stop_Active" )
      wire#w1
      R_Coil( "Pump3362_Xa_BonChua1" )
   END_RUNG
   RUNG wire#powerrail
      Contact( "PLC1_Loi_Tong" )
   END_RUNG wire#w1
   // the same network as SCL:
   IF "PLC1_Stop_Active" OR "PLC1_Loi_Tong" THEN "Pump3362_Xa_BonChua1" := FALSE; END_IF;
END_REGION

REGION Network 122: Dừng an toàn bồn chứa reset Pump3364_Filter khi Stop hoặc Lỗi tổng
   RUNG wire#powerrail
      Contact( "PLC1_Stop_Active" )
      wire#w1
      R_Coil( "Pump3364_Filter" )
   END_RUNG
   RUNG wire#powerrail
      Contact( "PLC1_Loi_Tong" )
   END_RUNG wire#w1
   // the same network as SCL:
   IF "PLC1_Stop_Active" OR "PLC1_Loi_Tong" THEN "Pump3364_Filter" := FALSE; END_IF;
END_REGION

REGION Network 123: Dừng an toàn bồn chứa reset Pump3365_Filter khi Stop hoặc Lỗi tổng
   RUNG wire#powerrail
      Contact( "PLC1_Stop_Active" )
      wire#w1
      R_Coil( "Pump3365_Filter" )
   END_RUNG
   RUNG wire#powerrail
      Contact( "PLC1_Loi_Tong" )
   END_RUNG wire#w1
   // the same network as SCL:
   IF "PLC1_Stop_Active" OR "PLC1_Loi_Tong" THEN "Pump3365_Filter" := FALSE; END_IF;
END_REGION

REGION Network 124: Dừng an toàn bồn chứa reset V3331_Xa_BonChua1 khi Stop hoặc Lỗi tổng
   RUNG wire#powerrail
      Contact( "PLC1_Stop_Active" )
      wire#w1
      R_Coil( "V3331_Xa_BonChua1" )
   END_RUNG
   RUNG wire#powerrail
      Contact( "PLC1_Loi_Tong" )
   END_RUNG wire#w1
   // the same network as SCL:
   IF "PLC1_Stop_Active" OR "PLC1_Loi_Tong" THEN "V3331_Xa_BonChua1" := FALSE; END_IF;
END_REGION

REGION Network 125: Dừng an toàn bồn chứa reset V3332_Xa_BonChua1 khi Stop hoặc Lỗi tổng
   RUNG wire#powerrail
      Contact( "PLC1_Stop_Active" )
      wire#w1
      R_Coil( "V3332_Xa_BonChua1" )
   END_RUNG
   RUNG wire#powerrail
      Contact( "PLC1_Loi_Tong" )
   END_RUNG wire#w1
   // the same network as SCL:
   IF "PLC1_Stop_Active" OR "PLC1_Loi_Tong" THEN "V3332_Xa_BonChua1" := FALSE; END_IF;
END_REGION

REGION Network 126: Dừng an toàn bồn chứa reset V3333_DieuHuong_BonChua1 khi Stop hoặc Lỗi tổng
   RUNG wire#powerrail
      Contact( "PLC1_Stop_Active" )
      wire#w1
      R_Coil( "V3333_DieuHuong_BonChua1" )
   END_RUNG
   RUNG wire#powerrail
      Contact( "PLC1_Loi_Tong" )
   END_RUNG wire#w1
   // the same network as SCL:
   IF "PLC1_Stop_Active" OR "PLC1_Loi_Tong" THEN "V3333_DieuHuong_BonChua1" := FALSE; END_IF;
END_REGION

REGION Network 127: Dừng an toàn bồn chứa reset V3334_DieuHuong_BonChua1 khi Stop hoặc Lỗi tổng
   RUNG wire#powerrail
      Contact( "PLC1_Stop_Active" )
      wire#w1
      R_Coil( "V3334_DieuHuong_BonChua1" )
   END_RUNG
   RUNG wire#powerrail
      Contact( "PLC1_Loi_Tong" )
   END_RUNG wire#w1
   // the same network as SCL:
   IF "PLC1_Stop_Active" OR "PLC1_Loi_Tong" THEN "V3334_DieuHuong_BonChua1" := FALSE; END_IF;
END_REGION

REGION Network 128: Dừng an toàn bồn chứa reset V3335_DieuHuong_BonChua1 khi Stop hoặc Lỗi tổng
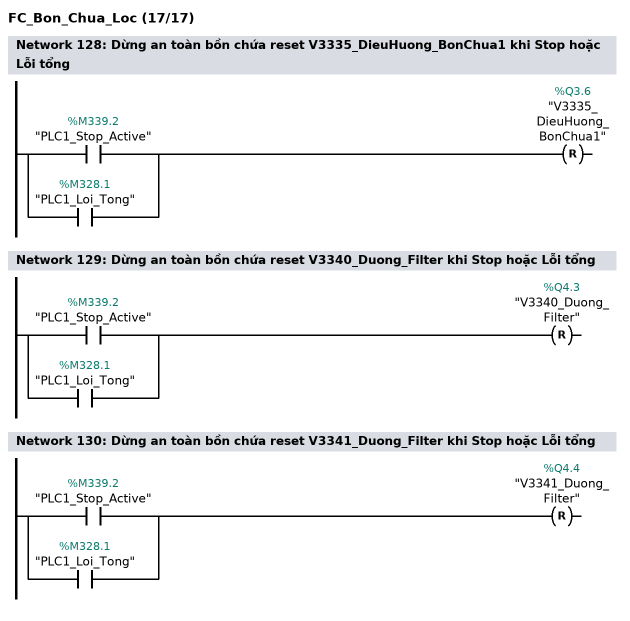
   RUNG wire#powerrail
      Contact( "PLC1_Stop_Active" )
      wire#w1
      R_Coil( "V3335_DieuHuong_BonChua1" )
   END_RUNG
   RUNG wire#powerrail
      Contact( "PLC1_Loi_Tong" )
   END_RUNG wire#w1
   // the same network as SCL:
   IF "PLC1_Stop_Active" OR "PLC1_Loi_Tong" THEN "V3335_DieuHuong_BonChua1" := FALSE; END_IF;
END_REGION

REGION Network 129: Dừng an toàn bồn chứa reset V3340_Duong_Filter khi Stop hoặc Lỗi tổng
   RUNG wire#powerrail
      Contact( "PLC1_Stop_Active" )
      wire#w1
      R_Coil( "V3340_Duong_Filter" )
   END_RUNG
   RUNG wire#powerrail
      Contact( "PLC1_Loi_Tong" )
   END_RUNG wire#w1
   // the same network as SCL:
   IF "PLC1_Stop_Active" OR "PLC1_Loi_Tong" THEN "V3340_Duong_Filter" := FALSE; END_IF;
END_REGION

REGION Network 130: Dừng an toàn bồn chứa reset V3341_Duong_Filter khi Stop hoặc Lỗi tổng
   RUNG wire#powerrail
      Contact( "PLC1_Stop_Active" )
      wire#w1
      R_Coil( "V3341_Duong_Filter" )
   END_RUNG
   RUNG wire#powerrail
      Contact( "PLC1_Loi_Tong" )
   END_RUNG wire#w1
   // the same network as SCL:
   IF "PLC1_Stop_Active" OR "PLC1_Loi_Tong" THEN "V3341_Duong_Filter" := FALSE; END_IF;
END_REGION
END_FUNCTION

FUNCTION "FC_Manual_Control_PLC1" : Void   // FC62, LAD
{ S7_Optimized_Access := 'TRUE' }
VERSION : 0.1
// stored: AutoNumber true, IsIECCheckEnabled false, SetENOAutomatically false, UDAEnableTagReadback false
BEGIN

REGION Network 1: Xác định trạng thái Manual Mode Active PLC1
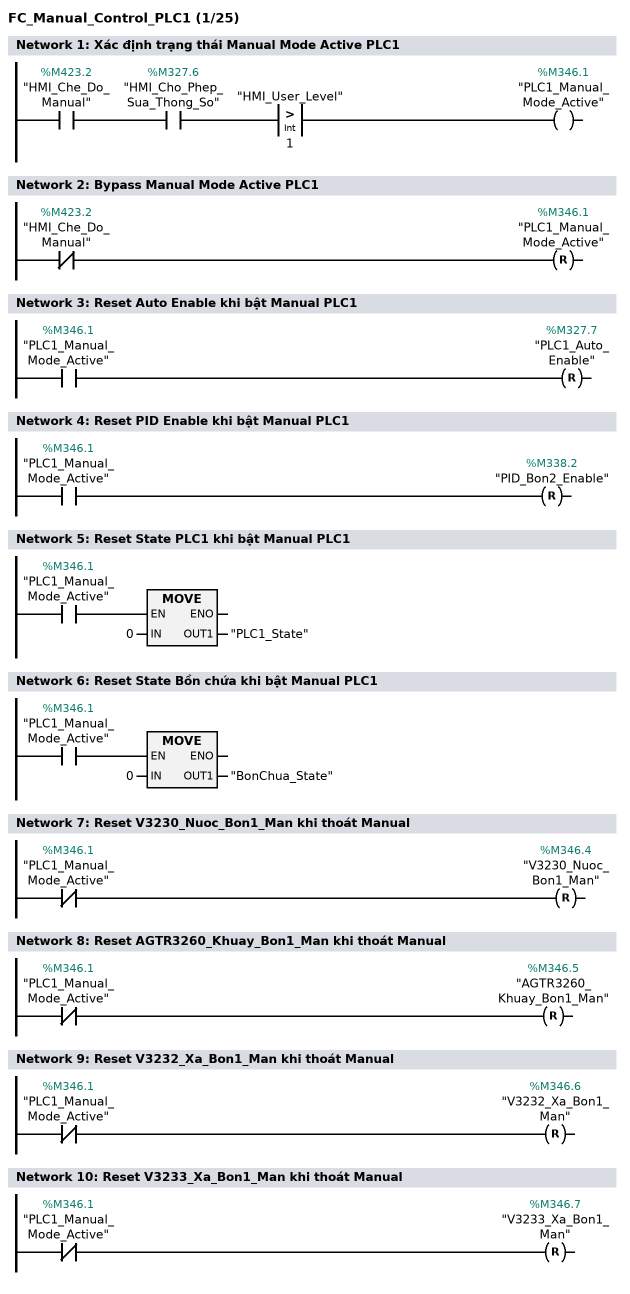
   RUNG wire#powerrail
      Contact( "HMI_Che_Do_Manual" )
      Contact( "HMI_Cho_Phep_Sua_Thong_So" )
      { S7_Templates := "SrcType := Int" } GT_Contact(in1 := "HMI_User_Level", in2 := 1)
      Coil( "PLC1_Manual_Mode_Active" )
   END_RUNG
   // the same network as SCL:
   "PLC1_Manual_Mode_Active" := "HMI_Che_Do_Manual" AND "HMI_Cho_Phep_Sua_Thong_So" AND ("HMI_User_Level" > 1);
END_REGION

REGION Network 2: Bypass Manual Mode Active PLC1
   RUNG wire#powerrail
      I_Contact( "HMI_Che_Do_Manual" )
      R_Coil( "PLC1_Manual_Mode_Active" )
   END_RUNG
   // the same network as SCL:
   IF NOT "HMI_Che_Do_Manual" THEN "PLC1_Manual_Mode_Active" := FALSE; END_IF;
END_REGION

REGION Network 3: Reset Auto Enable khi bật Manual PLC1
   RUNG wire#powerrail
      Contact( "PLC1_Manual_Mode_Active" )
      R_Coil( "PLC1_Auto_Enable" )
   END_RUNG
   // the same network as SCL:
   IF "PLC1_Manual_Mode_Active" THEN "PLC1_Auto_Enable" := FALSE; END_IF;
END_REGION

REGION Network 4: Reset PID Enable khi bật Manual PLC1
   RUNG wire#powerrail
      Contact( "PLC1_Manual_Mode_Active" )
      R_Coil( "PID_Bon2_Enable" )
   END_RUNG
   // the same network as SCL:
   IF "PLC1_Manual_Mode_Active" THEN "PID_Bon2_Enable" := FALSE; END_IF;
END_REGION

REGION Network 5: Reset State PLC1 khi bật Manual PLC1
   RUNG wire#powerrail
      Contact( "PLC1_Manual_Mode_Active" )
      { S7_GenerateENO := "TRUE" } Move(in := 0, out1 => "PLC1_State")
   END_RUNG
   // the same network as SCL:
   IF "PLC1_Manual_Mode_Active" THEN "PLC1_State" := 0; END_IF;
END_REGION

REGION Network 6: Reset State Bồn chứa khi bật Manual PLC1
   RUNG wire#powerrail
      Contact( "PLC1_Manual_Mode_Active" )
      { S7_GenerateENO := "TRUE" } Move(in := 0, out1 => "BonChua_State")
   END_RUNG
   // the same network as SCL:
   IF "PLC1_Manual_Mode_Active" THEN "BonChua_State" := 0; END_IF;
END_REGION

REGION Network 7: Reset V3230_Nuoc_Bon1_Man khi thoát Manual
   RUNG wire#powerrail
      I_Contact( "PLC1_Manual_Mode_Active" )
      R_Coil( "V3230_Nuoc_Bon1_Man" )
   END_RUNG
   // the same network as SCL:
   IF NOT "PLC1_Manual_Mode_Active" THEN "V3230_Nuoc_Bon1_Man" := FALSE; END_IF;
END_REGION

REGION Network 8: Reset AGTR3260_Khuay_Bon1_Man khi thoát Manual
   RUNG wire#powerrail
      I_Contact( "PLC1_Manual_Mode_Active" )
      R_Coil( "AGTR3260_Khuay_Bon1_Man" )
   END_RUNG
   // the same network as SCL:
   IF NOT "PLC1_Manual_Mode_Active" THEN "AGTR3260_Khuay_Bon1_Man" := FALSE; END_IF;
END_REGION

REGION Network 9: Reset V3232_Xa_Bon1_Man khi thoát Manual
   RUNG wire#powerrail
      I_Contact( "PLC1_Manual_Mode_Active" )
      R_Coil( "V3232_Xa_Bon1_Man" )
   END_RUNG
   // the same network as SCL:
   IF NOT "PLC1_Manual_Mode_Active" THEN "V3232_Xa_Bon1_Man" := FALSE; END_IF;
END_REGION

REGION Network 10: Reset V3233_Xa_Bon1_Man khi thoát Manual
   RUNG wire#powerrail
      I_Contact( "PLC1_Manual_Mode_Active" )
      R_Coil( "V3233_Xa_Bon1_Man" )
   END_RUNG
   // the same network as SCL:
   IF NOT "PLC1_Manual_Mode_Active" THEN "V3233_Xa_Bon1_Man" := FALSE; END_IF;
END_REGION

REGION Network 11: Reset V3234_Xa_Bon1_Man khi thoát Manual
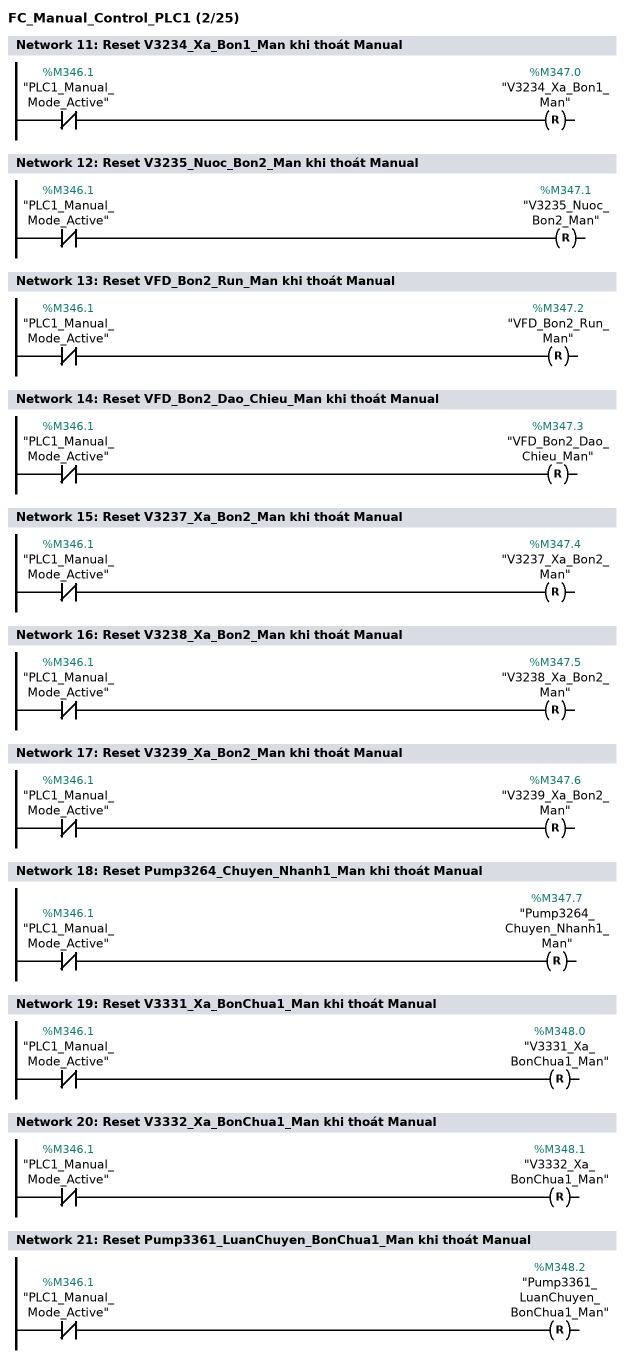
   RUNG wire#powerrail
      I_Contact( "PLC1_Manual_Mode_Active" )
      R_Coil( "V3234_Xa_Bon1_Man" )
   END_RUNG
   // the same network as SCL:
   IF NOT "PLC1_Manual_Mode_Active" THEN "V3234_Xa_Bon1_Man" := FALSE; END_IF;
END_REGION

REGION Network 12: Reset V3235_Nuoc_Bon2_Man khi thoát Manual
   RUNG wire#powerrail
      I_Contact( "PLC1_Manual_Mode_Active" )
      R_Coil( "V3235_Nuoc_Bon2_Man" )
   END_RUNG
   // the same network as SCL:
   IF NOT "PLC1_Manual_Mode_Active" THEN "V3235_Nuoc_Bon2_Man" := FALSE; END_IF;
END_REGION

REGION Network 13: Reset VFD_Bon2_Run_Man khi thoát Manual
   RUNG wire#powerrail
      I_Contact( "PLC1_Manual_Mode_Active" )
      R_Coil( "VFD_Bon2_Run_Man" )
   END_RUNG
   // the same network as SCL:
   IF NOT "PLC1_Manual_Mode_Active" THEN "VFD_Bon2_Run_Man" := FALSE; END_IF;
END_REGION

REGION Network 14: Reset VFD_Bon2_Dao_Chieu_Man khi thoát Manual
   RUNG wire#powerrail
      I_Contact( "PLC1_Manual_Mode_Active" )
      R_Coil( "VFD_Bon2_Dao_Chieu_Man" )
   END_RUNG
   // the same network as SCL:
   IF NOT "PLC1_Manual_Mode_Active" THEN "VFD_Bon2_Dao_Chieu_Man" := FALSE; END_IF;
END_REGION

REGION Network 15: Reset V3237_Xa_Bon2_Man khi thoát Manual
   RUNG wire#powerrail
      I_Contact( "PLC1_Manual_Mode_Active" )
      R_Coil( "V3237_Xa_Bon2_Man" )
   END_RUNG
   // the same network as SCL:
   IF NOT "PLC1_Manual_Mode_Active" THEN "V3237_Xa_Bon2_Man" := FALSE; END_IF;
END_REGION

REGION Network 16: Reset V3238_Xa_Bon2_Man khi thoát Manual
   RUNG wire#powerrail
      I_Contact( "PLC1_Manual_Mode_Active" )
      R_Coil( "V3238_Xa_Bon2_Man" )
   END_RUNG
   // the same network as SCL:
   IF NOT "PLC1_Manual_Mode_Active" THEN "V3238_Xa_Bon2_Man" := FALSE; END_IF;
END_REGION

REGION Network 17: Reset V3239_Xa_Bon2_Man khi thoát Manual
   RUNG wire#powerrail
      I_Contact( "PLC1_Manual_Mode_Active" )
      R_Coil( "V3239_Xa_Bon2_Man" )
   END_RUNG
   // the same network as SCL:
   IF NOT "PLC1_Manual_Mode_Active" THEN "V3239_Xa_Bon2_Man" := FALSE; END_IF;
END_REGION

REGION Network 18: Reset Pump3264_Chuyen_Nhanh1_Man khi thoát Manual
   RUNG wire#powerrail
      I_Contact( "PLC1_Manual_Mode_Active" )
      R_Coil( "Pump3264_Chuyen_Nhanh1_Man" )
   END_RUNG
   // the same network as SCL:
   IF NOT "PLC1_Manual_Mode_Active" THEN "Pump3264_Chuyen_Nhanh1_Man" := FALSE; END_IF;
END_REGION

REGION Network 19: Reset V3331_Xa_BonChua1_Man khi thoát Manual
   RUNG wire#powerrail
      I_Contact( "PLC1_Manual_Mode_Active" )
      R_Coil( "V3331_Xa_BonChua1_Man" )
   END_RUNG
   // the same network as SCL:
   IF NOT "PLC1_Manual_Mode_Active" THEN "V3331_Xa_BonChua1_Man" := FALSE; END_IF;
END_REGION

REGION Network 20: Reset V3332_Xa_BonChua1_Man khi thoát Manual
   RUNG wire#powerrail
      I_Contact( "PLC1_Manual_Mode_Active" )
      R_Coil( "V3332_Xa_BonChua1_Man" )
   END_RUNG
   // the same network as SCL:
   IF NOT "PLC1_Manual_Mode_Active" THEN "V3332_Xa_BonChua1_Man" := FALSE; END_IF;
END_REGION

REGION Network 21: Reset Pump3361_LuanChuyen_BonChua1_Man khi thoát Manual
   RUNG wire#powerrail
      I_Contact( "PLC1_Manual_Mode_Active" )
      R_Coil( "Pump3361_LuanChuyen_BonChua1_Man" )
   END_RUNG
   // the same network as SCL:
   IF NOT "PLC1_Manual_Mode_Active" THEN "Pump3361_LuanChuyen_BonChua1_Man" := FALSE; END_IF;
END_REGION

REGION Network 22: Reset Pump3362_Xa_BonChua1_Man khi thoát Manual
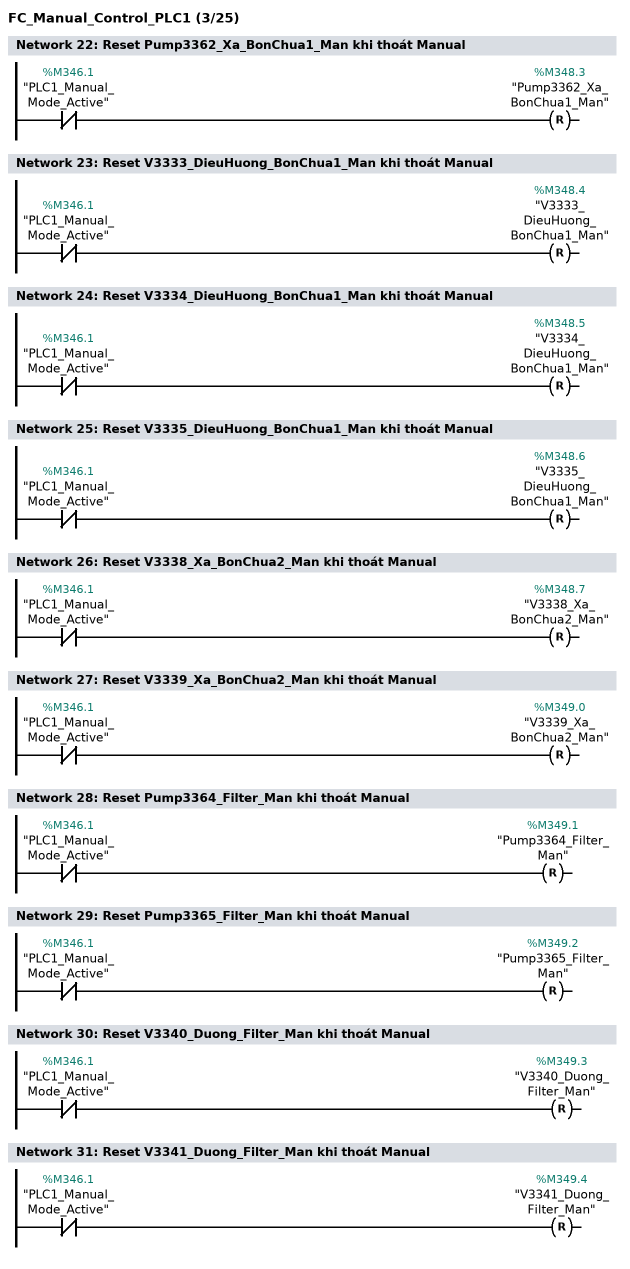
   RUNG wire#powerrail
      I_Contact( "PLC1_Manual_Mode_Active" )
      R_Coil( "Pump3362_Xa_BonChua1_Man" )
   END_RUNG
   // the same network as SCL:
   IF NOT "PLC1_Manual_Mode_Active" THEN "Pump3362_Xa_BonChua1_Man" := FALSE; END_IF;
END_REGION

REGION Network 23: Reset V3333_DieuHuong_BonChua1_Man khi thoát Manual
   RUNG wire#powerrail
      I_Contact( "PLC1_Manual_Mode_Active" )
      R_Coil( "V3333_DieuHuong_BonChua1_Man" )
   END_RUNG
   // the same network as SCL:
   IF NOT "PLC1_Manual_Mode_Active" THEN "V3333_DieuHuong_BonChua1_Man" := FALSE; END_IF;
END_REGION

REGION Network 24: Reset V3334_DieuHuong_BonChua1_Man khi thoát Manual
   RUNG wire#powerrail
      I_Contact( "PLC1_Manual_Mode_Active" )
      R_Coil( "V3334_DieuHuong_BonChua1_Man" )
   END_RUNG
   // the same network as SCL:
   IF NOT "PLC1_Manual_Mode_Active" THEN "V3334_DieuHuong_BonChua1_Man" := FALSE; END_IF;
END_REGION

REGION Network 25: Reset V3335_DieuHuong_BonChua1_Man khi thoát Manual
   RUNG wire#powerrail
      I_Contact( "PLC1_Manual_Mode_Active" )
      R_Coil( "V3335_DieuHuong_BonChua1_Man" )
   END_RUNG
   // the same network as SCL:
   IF NOT "PLC1_Manual_Mode_Active" THEN "V3335_DieuHuong_BonChua1_Man" := FALSE; END_IF;
END_REGION

REGION Network 26: Reset V3338_Xa_BonChua2_Man khi thoát Manual
   RUNG wire#powerrail
      I_Contact( "PLC1_Manual_Mode_Active" )
      R_Coil( "V3338_Xa_BonChua2_Man" )
   END_RUNG
   // the same network as SCL:
   IF NOT "PLC1_Manual_Mode_Active" THEN "V3338_Xa_BonChua2_Man" := FALSE; END_IF;
END_REGION

REGION Network 27: Reset V3339_Xa_BonChua2_Man khi thoát Manual
   RUNG wire#powerrail
      I_Contact( "PLC1_Manual_Mode_Active" )
      R_Coil( "V3339_Xa_BonChua2_Man" )
   END_RUNG
   // the same network as SCL:
   IF NOT "PLC1_Manual_Mode_Active" THEN "V3339_Xa_BonChua2_Man" := FALSE; END_IF;
END_REGION

REGION Network 28: Reset Pump3364_Filter_Man khi thoát Manual
   RUNG wire#powerrail
      I_Contact( "PLC1_Manual_Mode_Active" )
      R_Coil( "Pump3364_Filter_Man" )
   END_RUNG
   // the same network as SCL:
   IF NOT "PLC1_Manual_Mode_Active" THEN "Pump3364_Filter_Man" := FALSE; END_IF;
END_REGION

REGION Network 29: Reset Pump3365_Filter_Man khi thoát Manual
   RUNG wire#powerrail
      I_Contact( "PLC1_Manual_Mode_Active" )
      R_Coil( "Pump3365_Filter_Man" )
   END_RUNG
   // the same network as SCL:
   IF NOT "PLC1_Manual_Mode_Active" THEN "Pump3365_Filter_Man" := FALSE; END_IF;
END_REGION

REGION Network 30: Reset V3340_Duong_Filter_Man khi thoát Manual
   RUNG wire#powerrail
      I_Contact( "PLC1_Manual_Mode_Active" )
      R_Coil( "V3340_Duong_Filter_Man" )
   END_RUNG
   // the same network as SCL:
   IF NOT "PLC1_Manual_Mode_Active" THEN "V3340_Duong_Filter_Man" := FALSE; END_IF;
END_REGION

REGION Network 31: Reset V3341_Duong_Filter_Man khi thoát Manual
   RUNG wire#powerrail
      I_Contact( "PLC1_Manual_Mode_Active" )
      R_Coil( "V3341_Duong_Filter_Man" )
   END_RUNG
   // the same network as SCL:
   IF NOT "PLC1_Manual_Mode_Active" THEN "V3341_Duong_Filter_Man" := FALSE; END_IF;
END_REGION

REGION Network 32: Clear CV3201_Nuoc_Bon1_Man khi thoát Manual
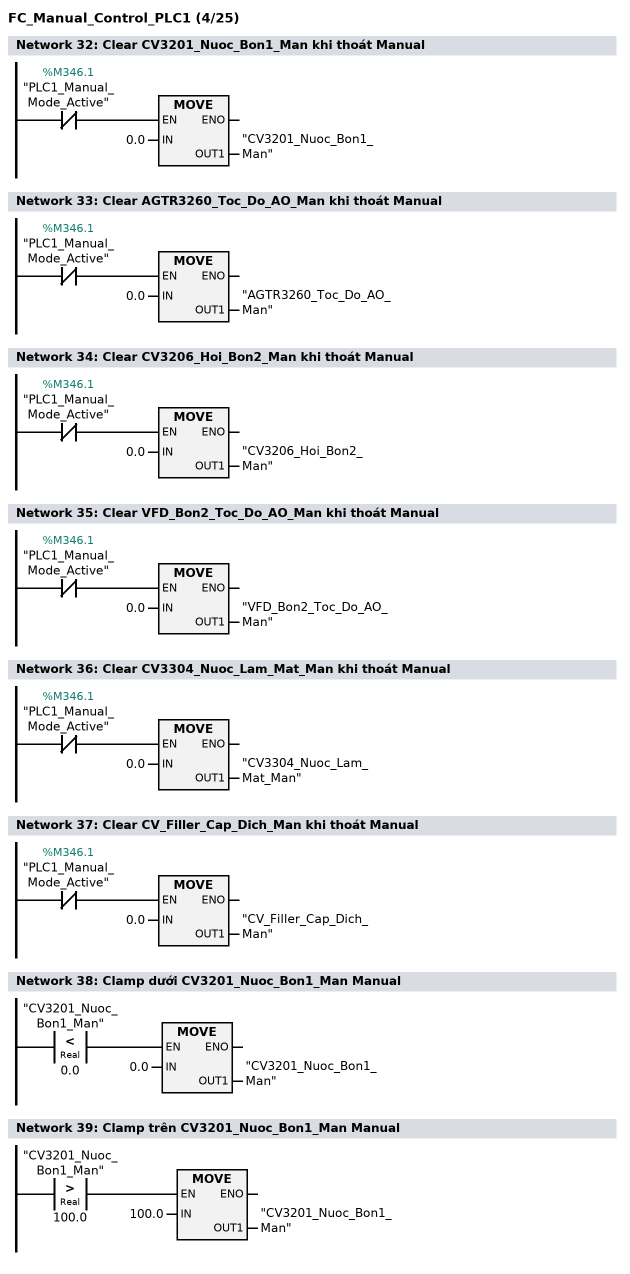
   RUNG wire#powerrail
      I_Contact( "PLC1_Manual_Mode_Active" )
      { S7_GenerateENO := "TRUE" } Move(in := 0.0, out1 => "CV3201_Nuoc_Bon1_Man")
   END_RUNG
   // the same network as SCL:
   IF NOT "PLC1_Manual_Mode_Active" THEN "CV3201_Nuoc_Bon1_Man" := 0.0; END_IF;
END_REGION

REGION Network 33: Clear AGTR3260_Toc_Do_AO_Man khi thoát Manual
   RUNG wire#powerrail
      I_Contact( "PLC1_Manual_Mode_Active" )
      { S7_GenerateENO := "TRUE" } Move(in := 0.0, out1 => "AGTR3260_Toc_Do_AO_Man")
   END_RUNG
   // the same network as SCL:
   IF NOT "PLC1_Manual_Mode_Active" THEN "AGTR3260_Toc_Do_AO_Man" := 0.0; END_IF;
END_REGION

REGION Network 34: Clear CV3206_Hoi_Bon2_Man khi thoát Manual
   RUNG wire#powerrail
      I_Contact( "PLC1_Manual_Mode_Active" )
      { S7_GenerateENO := "TRUE" } Move(in := 0.0, out1 => "CV3206_Hoi_Bon2_Man")
   END_RUNG
   // the same network as SCL:
   IF NOT "PLC1_Manual_Mode_Active" THEN "CV3206_Hoi_Bon2_Man" := 0.0; END_IF;
END_REGION

REGION Network 35: Clear VFD_Bon2_Toc_Do_AO_Man khi thoát Manual
   RUNG wire#powerrail
      I_Contact( "PLC1_Manual_Mode_Active" )
      { S7_GenerateENO := "TRUE" } Move(in := 0.0, out1 => "VFD_Bon2_Toc_Do_AO_Man")
   END_RUNG
   // the same network as SCL:
   IF NOT "PLC1_Manual_Mode_Active" THEN "VFD_Bon2_Toc_Do_AO_Man" := 0.0; END_IF;
END_REGION

REGION Network 36: Clear CV3304_Nuoc_Lam_Mat_Man khi thoát Manual
   RUNG wire#powerrail
      I_Contact( "PLC1_Manual_Mode_Active" )
      { S7_GenerateENO := "TRUE" } Move(in := 0.0, out1 => "CV3304_Nuoc_Lam_Mat_Man")
   END_RUNG
   // the same network as SCL:
   IF NOT "PLC1_Manual_Mode_Active" THEN "CV3304_Nuoc_Lam_Mat_Man" := 0.0; END_IF;
END_REGION

REGION Network 37: Clear CV_Filler_Cap_Dich_Man khi thoát Manual
   RUNG wire#powerrail
      I_Contact( "PLC1_Manual_Mode_Active" )
      { S7_GenerateENO := "TRUE" } Move(in := 0.0, out1 => "CV_Filler_Cap_Dich_Man")
   END_RUNG
   // the same network as SCL:
   IF NOT "PLC1_Manual_Mode_Active" THEN "CV_Filler_Cap_Dich_Man" := 0.0; END_IF;
END_REGION

REGION Network 38: Clamp dưới CV3201_Nuoc_Bon1_Man Manual
   RUNG wire#powerrail
      { S7_Templates := "SrcType := Real" } LT_Contact(in1 := "CV3201_Nuoc_Bon1_Man", in2 := 0.0)
      { S7_GenerateENO := "TRUE" } Move(in := 0.0, out1 => "CV3201_Nuoc_Bon1_Man")
   END_RUNG
   // the same network as SCL:
   IF "CV3201_Nuoc_Bon1_Man" < 0.0 THEN "CV3201_Nuoc_Bon1_Man" := 0.0; END_IF;
END_REGION

REGION Network 39: Clamp trên CV3201_Nuoc_Bon1_Man Manual
   RUNG wire#powerrail
      { S7_Templates := "SrcType := Real" } GT_Contact(in1 := "CV3201_Nuoc_Bon1_Man", in2 := 100.0)
      { S7_GenerateENO := "TRUE" } Move(in := 100.0, out1 => "CV3201_Nuoc_Bon1_Man")
   END_RUNG
   // the same network as SCL:
   IF "CV3201_Nuoc_Bon1_Man" > 100.0 THEN "CV3201_Nuoc_Bon1_Man" := 100.0; END_IF;
END_REGION

REGION Network 40: Clamp dưới AGTR3260_Toc_Do_AO_Man Manual
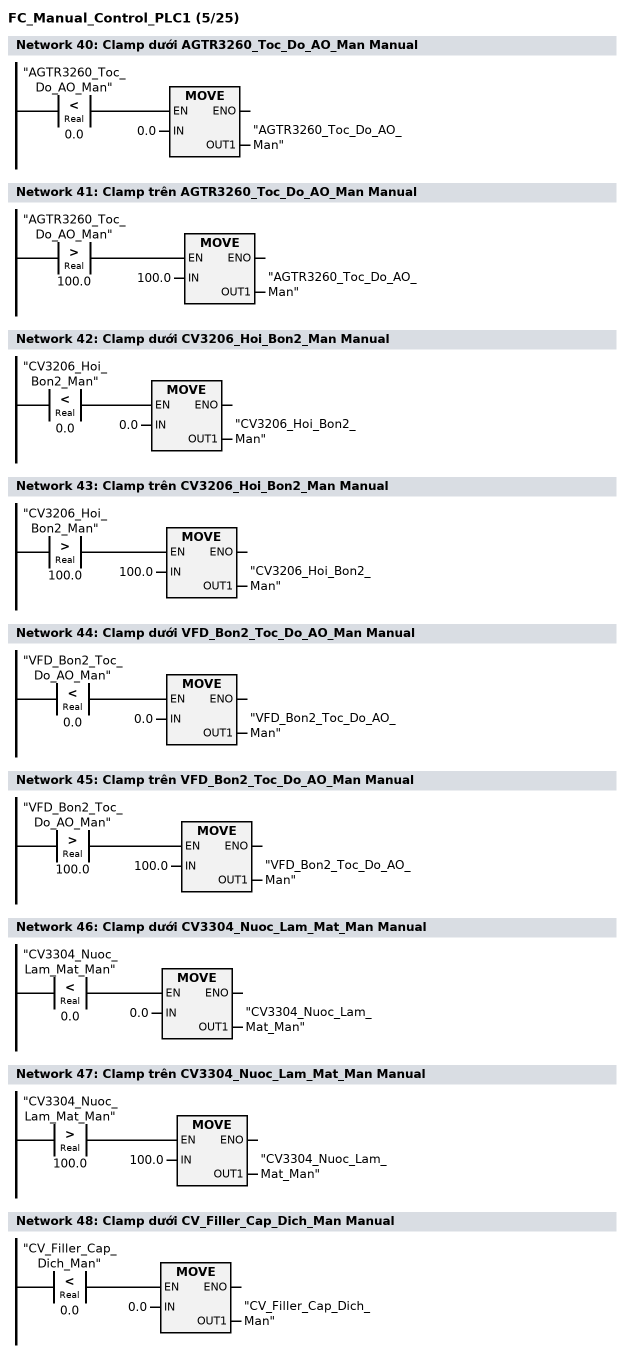
   RUNG wire#powerrail
      { S7_Templates := "SrcType := Real" } LT_Contact(in1 := "AGTR3260_Toc_Do_AO_Man", in2 := 0.0)
      { S7_GenerateENO := "TRUE" } Move(in := 0.0, out1 => "AGTR3260_Toc_Do_AO_Man")
   END_RUNG
   // the same network as SCL:
   IF "AGTR3260_Toc_Do_AO_Man" < 0.0 THEN "AGTR3260_Toc_Do_AO_Man" := 0.0; END_IF;
END_REGION

REGION Network 41: Clamp trên AGTR3260_Toc_Do_AO_Man Manual
   RUNG wire#powerrail
      { S7_Templates := "SrcType := Real" } GT_Contact(in1 := "AGTR3260_Toc_Do_AO_Man", in2 := 100.0)
      { S7_GenerateENO := "TRUE" } Move(in := 100.0, out1 => "AGTR3260_Toc_Do_AO_Man")
   END_RUNG
   // the same network as SCL:
   IF "AGTR3260_Toc_Do_AO_Man" > 100.0 THEN "AGTR3260_Toc_Do_AO_Man" := 100.0; END_IF;
END_REGION

REGION Network 42: Clamp dưới CV3206_Hoi_Bon2_Man Manual
   RUNG wire#powerrail
      { S7_Templates := "SrcType := Real" } LT_Contact(in1 := "CV3206_Hoi_Bon2_Man", in2 := 0.0)
      { S7_GenerateENO := "TRUE" } Move(in := 0.0, out1 => "CV3206_Hoi_Bon2_Man")
   END_RUNG
   // the same network as SCL:
   IF "CV3206_Hoi_Bon2_Man" < 0.0 THEN "CV3206_Hoi_Bon2_Man" := 0.0; END_IF;
END_REGION

REGION Network 43: Clamp trên CV3206_Hoi_Bon2_Man Manual
   RUNG wire#powerrail
      { S7_Templates := "SrcType := Real" } GT_Contact(in1 := "CV3206_Hoi_Bon2_Man", in2 := 100.0)
      { S7_GenerateENO := "TRUE" } Move(in := 100.0, out1 => "CV3206_Hoi_Bon2_Man")
   END_RUNG
   // the same network as SCL:
   IF "CV3206_Hoi_Bon2_Man" > 100.0 THEN "CV3206_Hoi_Bon2_Man" := 100.0; END_IF;
END_REGION

REGION Network 44: Clamp dưới VFD_Bon2_Toc_Do_AO_Man Manual
   RUNG wire#powerrail
      { S7_Templates := "SrcType := Real" } LT_Contact(in1 := "VFD_Bon2_Toc_Do_AO_Man", in2 := 0.0)
      { S7_GenerateENO := "TRUE" } Move(in := 0.0, out1 => "VFD_Bon2_Toc_Do_AO_Man")
   END_RUNG
   // the same network as SCL:
   IF "VFD_Bon2_Toc_Do_AO_Man" < 0.0 THEN "VFD_Bon2_Toc_Do_AO_Man" := 0.0; END_IF;
END_REGION

REGION Network 45: Clamp trên VFD_Bon2_Toc_Do_AO_Man Manual
   RUNG wire#powerrail
      { S7_Templates := "SrcType := Real" } GT_Contact(in1 := "VFD_Bon2_Toc_Do_AO_Man", in2 := 100.0)
      { S7_GenerateENO := "TRUE" } Move(in := 100.0, out1 => "VFD_Bon2_Toc_Do_AO_Man")
   END_RUNG
   // the same network as SCL:
   IF "VFD_Bon2_Toc_Do_AO_Man" > 100.0 THEN "VFD_Bon2_Toc_Do_AO_Man" := 100.0; END_IF;
END_REGION

REGION Network 46: Clamp dưới CV3304_Nuoc_Lam_Mat_Man Manual
   RUNG wire#powerrail
      { S7_Templates := "SrcType := Real" } LT_Contact(in1 := "CV3304_Nuoc_Lam_Mat_Man", in2 := 0.0)
      { S7_GenerateENO := "TRUE" } Move(in := 0.0, out1 => "CV3304_Nuoc_Lam_Mat_Man")
   END_RUNG
   // the same network as SCL:
   IF "CV3304_Nuoc_Lam_Mat_Man" < 0.0 THEN "CV3304_Nuoc_Lam_Mat_Man" := 0.0; END_IF;
END_REGION

REGION Network 47: Clamp trên CV3304_Nuoc_Lam_Mat_Man Manual
   RUNG wire#powerrail
      { S7_Templates := "SrcType := Real" } GT_Contact(in1 := "CV3304_Nuoc_Lam_Mat_Man", in2 := 100.0)
      { S7_GenerateENO := "TRUE" } Move(in := 100.0, out1 => "CV3304_Nuoc_Lam_Mat_Man")
   END_RUNG
   // the same network as SCL:
   IF "CV3304_Nuoc_Lam_Mat_Man" > 100.0 THEN "CV3304_Nuoc_Lam_Mat_Man" := 100.0; END_IF;
END_REGION

REGION Network 48: Clamp dưới CV_Filler_Cap_Dich_Man Manual
   RUNG wire#powerrail
      { S7_Templates := "SrcType := Real" } LT_Contact(in1 := "CV_Filler_Cap_Dich_Man", in2 := 0.0)
      { S7_GenerateENO := "TRUE" } Move(in := 0.0, out1 => "CV_Filler_Cap_Dich_Man")
   END_RUNG
   // the same network as SCL:
   IF "CV_Filler_Cap_Dich_Man" < 0.0 THEN "CV_Filler_Cap_Dich_Man" := 0.0; END_IF;
END_REGION

REGION Network 49: Clamp trên CV_Filler_Cap_Dich_Man Manual
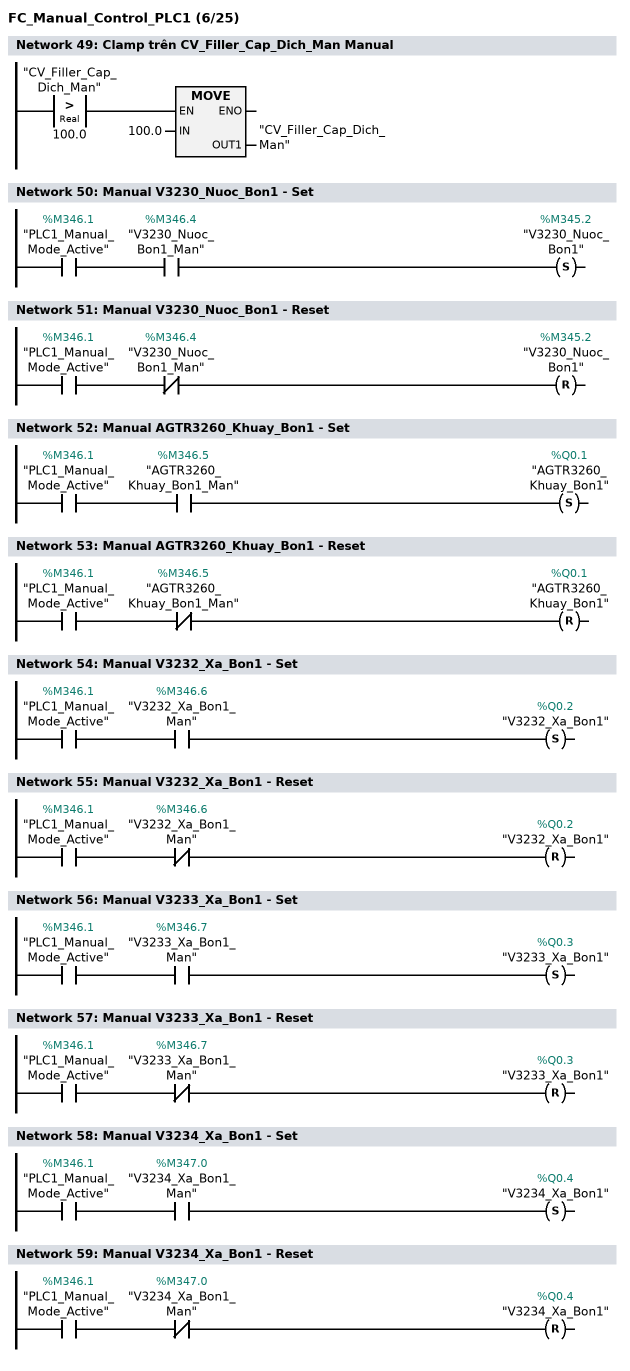
   RUNG wire#powerrail
      { S7_Templates := "SrcType := Real" } GT_Contact(in1 := "CV_Filler_Cap_Dich_Man", in2 := 100.0)
      { S7_GenerateENO := "TRUE" } Move(in := 100.0, out1 => "CV_Filler_Cap_Dich_Man")
   END_RUNG
   // the same network as SCL:
   IF "CV_Filler_Cap_Dich_Man" > 100.0 THEN "CV_Filler_Cap_Dich_Man" := 100.0; END_IF;
END_REGION

REGION Network 50: Manual V3230_Nuoc_Bon1 - Set
   RUNG wire#powerrail
      Contact( "PLC1_Manual_Mode_Active" )
      Contact( "V3230_Nuoc_Bon1_Man" )
      S_Coil( "V3230_Nuoc_Bon1" )
   END_RUNG
   // the same network as SCL:
   IF "PLC1_Manual_Mode_Active" AND "V3230_Nuoc_Bon1_Man" THEN "V3230_Nuoc_Bon1" := TRUE; END_IF;
END_REGION

REGION Network 51: Manual V3230_Nuoc_Bon1 - Reset
   RUNG wire#powerrail
      Contact( "PLC1_Manual_Mode_Active" )
      I_Contact( "V3230_Nuoc_Bon1_Man" )
      R_Coil( "V3230_Nuoc_Bon1" )
   END_RUNG
   // the same network as SCL:
   IF "PLC1_Manual_Mode_Active" AND NOT "V3230_Nuoc_Bon1_Man" THEN "V3230_Nuoc_Bon1" := FALSE; END_IF;
END_REGION

REGION Network 52: Manual AGTR3260_Khuay_Bon1 - Set
   RUNG wire#powerrail
      Contact( "PLC1_Manual_Mode_Active" )
      Contact( "AGTR3260_Khuay_Bon1_Man" )
      S_Coil( "AGTR3260_Khuay_Bon1" )
   END_RUNG
   // the same network as SCL:
   IF "PLC1_Manual_Mode_Active" AND "AGTR3260_Khuay_Bon1_Man" THEN "AGTR3260_Khuay_Bon1" := TRUE; END_IF;
END_REGION

REGION Network 53: Manual AGTR3260_Khuay_Bon1 - Reset
   RUNG wire#powerrail
      Contact( "PLC1_Manual_Mode_Active" )
      I_Contact( "AGTR3260_Khuay_Bon1_Man" )
      R_Coil( "AGTR3260_Khuay_Bon1" )
   END_RUNG
   // the same network as SCL:
   IF "PLC1_Manual_Mode_Active" AND NOT "AGTR3260_Khuay_Bon1_Man" THEN
       "AGTR3260_Khuay_Bon1" := FALSE;
   END_IF;
END_REGION

REGION Network 54: Manual V3232_Xa_Bon1 - Set
   RUNG wire#powerrail
      Contact( "PLC1_Manual_Mode_Active" )
      Contact( "V3232_Xa_Bon1_Man" )
      S_Coil( "V3232_Xa_Bon1" )
   END_RUNG
   // the same network as SCL:
   IF "PLC1_Manual_Mode_Active" AND "V3232_Xa_Bon1_Man" THEN "V3232_Xa_Bon1" := TRUE; END_IF;
END_REGION

REGION Network 55: Manual V3232_Xa_Bon1 - Reset
   RUNG wire#powerrail
      Contact( "PLC1_Manual_Mode_Active" )
      I_Contact( "V3232_Xa_Bon1_Man" )
      R_Coil( "V3232_Xa_Bon1" )
   END_RUNG
   // the same network as SCL:
   IF "PLC1_Manual_Mode_Active" AND NOT "V3232_Xa_Bon1_Man" THEN "V3232_Xa_Bon1" := FALSE; END_IF;
END_REGION

REGION Network 56: Manual V3233_Xa_Bon1 - Set
   RUNG wire#powerrail
      Contact( "PLC1_Manual_Mode_Active" )
      Contact( "V3233_Xa_Bon1_Man" )
      S_Coil( "V3233_Xa_Bon1" )
   END_RUNG
   // the same network as SCL:
   IF "PLC1_Manual_Mode_Active" AND "V3233_Xa_Bon1_Man" THEN "V3233_Xa_Bon1" := TRUE; END_IF;
END_REGION

REGION Network 57: Manual V3233_Xa_Bon1 - Reset
   RUNG wire#powerrail
      Contact( "PLC1_Manual_Mode_Active" )
      I_Contact( "V3233_Xa_Bon1_Man" )
      R_Coil( "V3233_Xa_Bon1" )
   END_RUNG
   // the same network as SCL:
   IF "PLC1_Manual_Mode_Active" AND NOT "V3233_Xa_Bon1_Man" THEN "V3233_Xa_Bon1" := FALSE; END_IF;
END_REGION

REGION Network 58: Manual V3234_Xa_Bon1 - Set
   RUNG wire#powerrail
      Contact( "PLC1_Manual_Mode_Active" )
      Contact( "V3234_Xa_Bon1_Man" )
      S_Coil( "V3234_Xa_Bon1" )
   END_RUNG
   // the same network as SCL:
   IF "PLC1_Manual_Mode_Active" AND "V3234_Xa_Bon1_Man" THEN "V3234_Xa_Bon1" := TRUE; END_IF;
END_REGION

REGION Network 59: Manual V3234_Xa_Bon1 - Reset
   RUNG wire#powerrail
      Contact( "PLC1_Manual_Mode_Active" )
      I_Contact( "V3234_Xa_Bon1_Man" )
      R_Coil( "V3234_Xa_Bon1" )
   END_RUNG
   // the same network as SCL:
   IF "PLC1_Manual_Mode_Active" AND NOT "V3234_Xa_Bon1_Man" THEN "V3234_Xa_Bon1" := FALSE; END_IF;
END_REGION

REGION Network 60: Manual V3235_Nuoc_Bon2 - Set
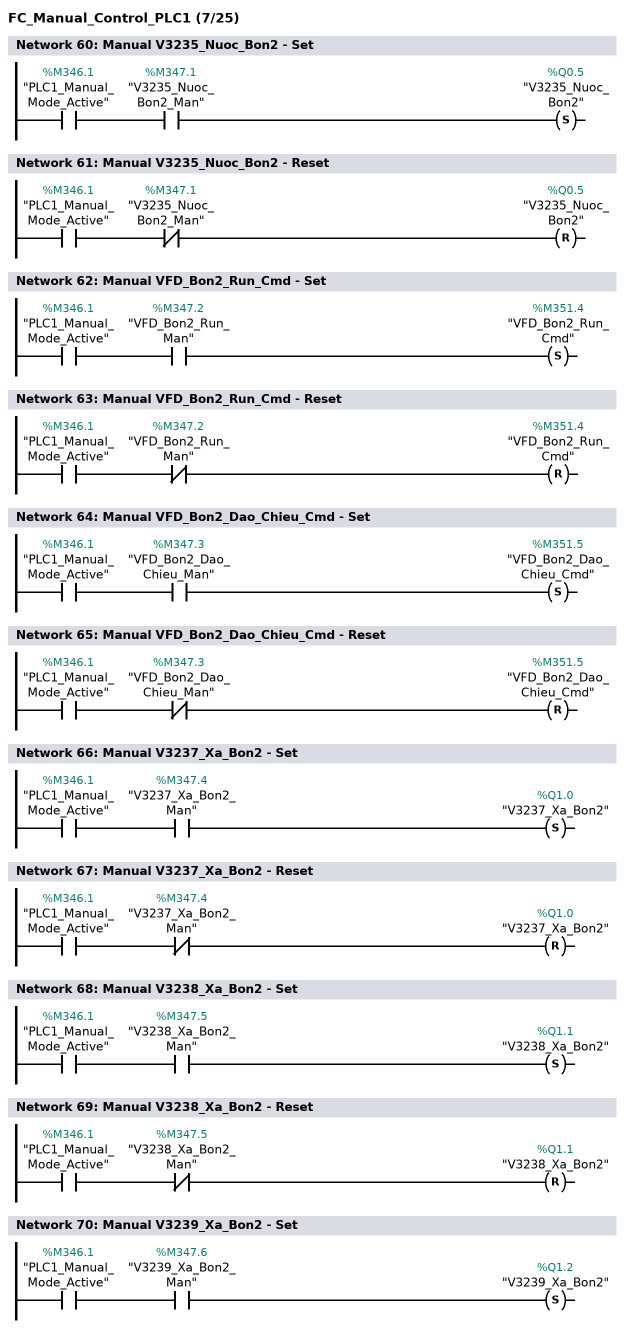
   RUNG wire#powerrail
      Contact( "PLC1_Manual_Mode_Active" )
      Contact( "V3235_Nuoc_Bon2_Man" )
      S_Coil( "V3235_Nuoc_Bon2" )
   END_RUNG
   // the same network as SCL:
   IF "PLC1_Manual_Mode_Active" AND "V3235_Nuoc_Bon2_Man" THEN "V3235_Nuoc_Bon2" := TRUE; END_IF;
END_REGION

REGION Network 61: Manual V3235_Nuoc_Bon2 - Reset
   RUNG wire#powerrail
      Contact( "PLC1_Manual_Mode_Active" )
      I_Contact( "V3235_Nuoc_Bon2_Man" )
      R_Coil( "V3235_Nuoc_Bon2" )
   END_RUNG
   // the same network as SCL:
   IF "PLC1_Manual_Mode_Active" AND NOT "V3235_Nuoc_Bon2_Man" THEN "V3235_Nuoc_Bon2" := FALSE; END_IF;
END_REGION

REGION Network 62: Manual VFD_Bon2_Run_Cmd - Set
   RUNG wire#powerrail
      Contact( "PLC1_Manual_Mode_Active" )
      Contact( "VFD_Bon2_Run_Man" )
      S_Coil( "VFD_Bon2_Run_Cmd" )
   END_RUNG
   // the same network as SCL:
   IF "PLC1_Manual_Mode_Active" AND "VFD_Bon2_Run_Man" THEN "VFD_Bon2_Run_Cmd" := TRUE; END_IF;
END_REGION

REGION Network 63: Manual VFD_Bon2_Run_Cmd - Reset
   RUNG wire#powerrail
      Contact( "PLC1_Manual_Mode_Active" )
      I_Contact( "VFD_Bon2_Run_Man" )
      R_Coil( "VFD_Bon2_Run_Cmd" )
   END_RUNG
   // the same network as SCL:
   IF "PLC1_Manual_Mode_Active" AND NOT "VFD_Bon2_Run_Man" THEN "VFD_Bon2_Run_Cmd" := FALSE; END_IF;
END_REGION

REGION Network 64: Manual VFD_Bon2_Dao_Chieu_Cmd - Set
   RUNG wire#powerrail
      Contact( "PLC1_Manual_Mode_Active" )
      Contact( "VFD_Bon2_Dao_Chieu_Man" )
      S_Coil( "VFD_Bon2_Dao_Chieu_Cmd" )
   END_RUNG
   // the same network as SCL:
   IF "PLC1_Manual_Mode_Active" AND "VFD_Bon2_Dao_Chieu_Man" THEN "VFD_Bon2_Dao_Chieu_Cmd" := TRUE; END_IF;
END_REGION

REGION Network 65: Manual VFD_Bon2_Dao_Chieu_Cmd - Reset
   RUNG wire#powerrail
      Contact( "PLC1_Manual_Mode_Active" )
      I_Contact( "VFD_Bon2_Dao_Chieu_Man" )
      R_Coil( "VFD_Bon2_Dao_Chieu_Cmd" )
   END_RUNG
   // the same network as SCL:
   IF "PLC1_Manual_Mode_Active" AND NOT "VFD_Bon2_Dao_Chieu_Man" THEN
       "VFD_Bon2_Dao_Chieu_Cmd" := FALSE;
   END_IF;
END_REGION

REGION Network 66: Manual V3237_Xa_Bon2 - Set
   RUNG wire#powerrail
      Contact( "PLC1_Manual_Mode_Active" )
      Contact( "V3237_Xa_Bon2_Man" )
      S_Coil( "V3237_Xa_Bon2" )
   END_RUNG
   // the same network as SCL:
   IF "PLC1_Manual_Mode_Active" AND "V3237_Xa_Bon2_Man" THEN "V3237_Xa_Bon2" := TRUE; END_IF;
END_REGION

REGION Network 67: Manual V3237_Xa_Bon2 - Reset
   RUNG wire#powerrail
      Contact( "PLC1_Manual_Mode_Active" )
      I_Contact( "V3237_Xa_Bon2_Man" )
      R_Coil( "V3237_Xa_Bon2" )
   END_RUNG
   // the same network as SCL:
   IF "PLC1_Manual_Mode_Active" AND NOT "V3237_Xa_Bon2_Man" THEN "V3237_Xa_Bon2" := FALSE; END_IF;
END_REGION

REGION Network 68: Manual V3238_Xa_Bon2 - Set
   RUNG wire#powerrail
      Contact( "PLC1_Manual_Mode_Active" )
      Contact( "V3238_Xa_Bon2_Man" )
      S_Coil( "V3238_Xa_Bon2" )
   END_RUNG
   // the same network as SCL:
   IF "PLC1_Manual_Mode_Active" AND "V3238_Xa_Bon2_Man" THEN "V3238_Xa_Bon2" := TRUE; END_IF;
END_REGION

REGION Network 69: Manual V3238_Xa_Bon2 - Reset
   RUNG wire#powerrail
      Contact( "PLC1_Manual_Mode_Active" )
      I_Contact( "V3238_Xa_Bon2_Man" )
      R_Coil( "V3238_Xa_Bon2" )
   END_RUNG
   // the same network as SCL:
   IF "PLC1_Manual_Mode_Active" AND NOT "V3238_Xa_Bon2_Man" THEN "V3238_Xa_Bon2" := FALSE; END_IF;
END_REGION

REGION Network 70: Manual V3239_Xa_Bon2 - Set
   RUNG wire#powerrail
      Contact( "PLC1_Manual_Mode_Active" )
      Contact( "V3239_Xa_Bon2_Man" )
      S_Coil( "V3239_Xa_Bon2" )
   END_RUNG
   // the same network as SCL:
   IF "PLC1_Manual_Mode_Active" AND "V3239_Xa_Bon2_Man" THEN "V3239_Xa_Bon2" := TRUE; END_IF;
END_REGION

REGION Network 71: Manual V3239_Xa_Bon2 - Reset
